REGION Network 26: U201 - ROTAZIONE + CM
   // "U201_OFF1"/"U201_OFF3"
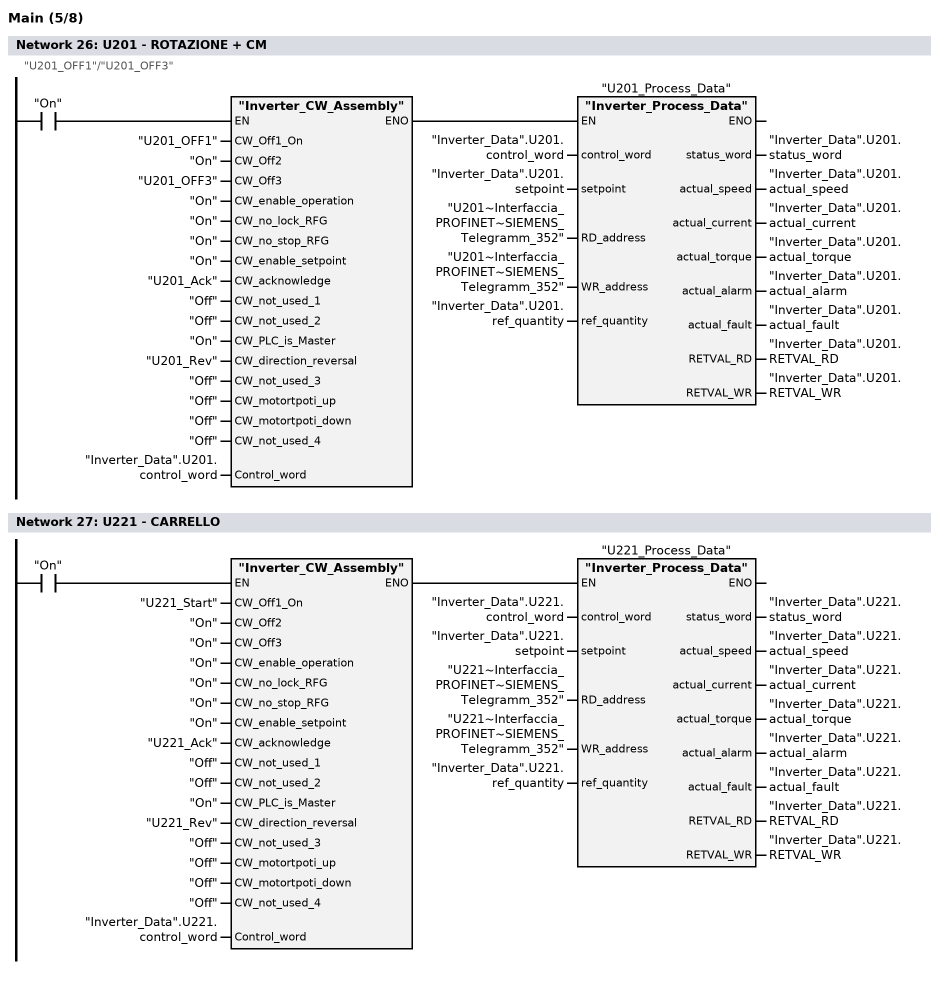
   RUNG wire#powerrail
      Contact( "On" )
      "Inverter_CW_Assembly"(CW_Off1_On := "U201_OFF1", CW_Off2 := "On", CW_Off3 := "U201_OFF3", CW_enable_operation := "On", CW_no_lock_RFG := "On", CW_no_stop_RFG := "On", CW_enable_setpoint := "On", CW_acknowledge := "U201_Ack", CW_not_used_1 := "Off", CW_not_used_2 := "Off", CW_PLC_is_Master := "On", CW_direction_reversal := "U201_Rev", CW_not_used_3 := "Off", CW_motortpoti_up := "Off", CW_motortpoti_down := "Off", CW_not_used_4 := "Off", Control_word := "Inverter_Data".U201.control_word)
      "U201_Process_Data"(control_word := "Inverter_Data".U201.control_word, setpoint := "Inverter_Data".U201.setpoint, RD_address := "U201~Interfaccia_PROFINET~SIEMENS_Telegramm_352", WR_address := "U201~Interfaccia_PROFINET~SIEMENS_Telegramm_352", ref_quantity := "Inverter_Data".U201.ref_quantity, status_word => "Inverter_Data".U201.status_word, actual_speed => "Inverter_Data".U201.actual_speed, actual_current => "Inverter_Data".U201.actual_current, actual_torque => "Inverter_Data".U201.actual_torque, actual_alarm => "Inverter_Data".U201.actual_alarm, actual_fault => "Inverter_Data".U201.actual_fault, RETVAL_RD => "Inverter_Data".U201.RETVAL_RD, RETVAL_WR => "Inverter_Data".U201.RETVAL_WR)
   END_RUNG
   // the same network as SCL:
   "Inverter_CW_Assembly"(EN := "On",
                          CW_Off1_On := "U201_OFF1",
                          CW_Off2 := "On",
                          CW_Off3 := "U201_OFF3",
                          CW_enable_operation := "On",
                          CW_no_lock_RFG := "On",
                          CW_no_stop_RFG := "On",
                          CW_enable_setpoint := "On",
                          CW_acknowledge := "U201_Ack",
                          CW_not_used_1 := "Off",
                          CW_not_used_2 := "Off",
                          CW_PLC_is_Master := "On",
                          CW_direction_reversal := "U201_Rev",
                          CW_not_used_3 := "Off",
                          CW_motortpoti_up := "Off",
                          CW_motortpoti_down := "Off",
                          CW_not_used_4 := "Off",
                          Control_word := "Inverter_Data".U201.control_word,
                          ENO => #_w1);
   IF #_w1 THEN
       "U201_Process_Data"(control_word := "Inverter_Data".U201.control_word,   // "Inverter_Process_Data"
                           setpoint := "Inverter_Data".U201.setpoint,
                           RD_address := "U201~Interfaccia_PROFINET~SIEMENS_Telegramm_352",
                           WR_address := "U201~Interfaccia_PROFINET~SIEMENS_Telegramm_352",
                           ref_quantity := "Inverter_Data".U201.ref_quantity,
                           status_word => "Inverter_Data".U201.status_word,
                           actual_speed => "Inverter_Data".U201.actual_speed,
                           actual_current => "Inverter_Data".U201.actual_current,
                           actual_torque => "Inverter_Data".U201.actual_torque,
                           actual_alarm => "Inverter_Data".U201.actual_alarm,
                           actual_fault => "Inverter_Data".U201.actual_fault,
                           RETVAL_RD => "Inverter_Data".U201.RETVAL_RD,
                           RETVAL_WR => "Inverter_Data".U201.RETVAL_WR);
   END_IF;
END_REGION

REGION Network 27: U221 - CARRELLO
   RUNG wire#powerrail
      Contact( "On" )
      "Inverter_CW_Assembly"(CW_Off1_On := "U221_Start", CW_Off2 := "On", CW_Off3 := "On", CW_enable_operation := "On", CW_no_lock_RFG := "On", CW_no_stop_RFG := "On", CW_enable_setpoint := "On", CW_acknowledge := "U221_Ack", CW_not_used_1 := "Off", CW_not_used_2 := "Off", CW_PLC_is_Master := "On", CW_direction_reversal := "U221_Rev", CW_not_used_3 := "Off", CW_motortpoti_up := "Off", CW_motortpoti_down := "Off", CW_not_used_4 := "Off", Control_word := "Inverter_Data".U221.control_word)
      "U221_Process_Data"(control_word := "Inverter_Data".U221.control_word, setpoint := "Inverter_Data".U221.setpoint, RD_address := "U221~Interfaccia_PROFINET~SIEMENS_Telegramm_352", WR_address := "U221~Interfaccia_PROFINET~SIEMENS_Telegramm_352", ref_quantity := "Inverter_Data".U221.ref_quantity, status_word => "Inverter_Data".U221.status_word, actual_speed => "Inverter_Data".U221.actual_speed, actual_current => "Inverter_Data".U221.actual_current, actual_torque => "Inverter_Data".U221.actual_torque, actual_alarm => "Inverter_Data".U221.actual_alarm, actual_fault => "Inverter_Data".U221.actual_fault, RETVAL_RD => "Inverter_Data".U221.RETVAL_RD, RETVAL_WR => "Inverter_Data".U221.RETVAL_WR)
   END_RUNG
   // the same network as SCL:
   "Inverter_CW_Assembly"(EN := "On",
                          CW_Off1_On := "U221_Start",
                          CW_Off2 := "On",
                          CW_Off3 := "On",
                          CW_enable_operation := "On",
                          CW_no_lock_RFG := "On",
                          CW_no_stop_RFG := "On",
                          CW_enable_setpoint := "On",
                          CW_acknowledge := "U221_Ack",
                          CW_not_used_1 := "Off",
                          CW_not_used_2 := "Off",
                          CW_PLC_is_Master := "On",
                          CW_direction_reversal := "U221_Rev",
                          CW_not_used_3 := "Off",
                          CW_motortpoti_up := "Off",
                          CW_motortpoti_down := "Off",
                          CW_not_used_4 := "Off",
                          Control_word := "Inverter_Data".U221.control_word,
                          ENO => #_w1);
   IF #_w1 THEN
       "U221_Process_Data"(control_word := "Inverter_Data".U221.control_word,   // "Inverter_Process_Data"
                           setpoint := "Inverter_Data".U221.setpoint,
                           RD_address := "U221~Interfaccia_PROFINET~SIEMENS_Telegramm_352",
                           WR_address := "U221~Interfaccia_PROFINET~SIEMENS_Telegramm_352",
                           ref_quantity := "Inverter_Data".U221.ref_quantity,
                           status_word => "Inverter_Data".U221.status_word,
                           actual_speed => "Inverter_Data".U221.actual_speed,
                           actual_current => "Inverter_Data".U221.actual_current,
                           actual_torque => "Inverter_Data".U221.actual_torque,
                           actual_alarm => "Inverter_Data".U221.actual_alarm,
                           actual_fault => "Inverter_Data".U221.actual_fault,
                           RETVAL_RD => "Inverter_Data".U221.RETVAL_RD,
                           RETVAL_WR => "Inverter_Data".U221.RETVAL_WR);
   END_IF;
END_REGION

REGION Network 28: U241 - PRESTIRO (VELOCE)
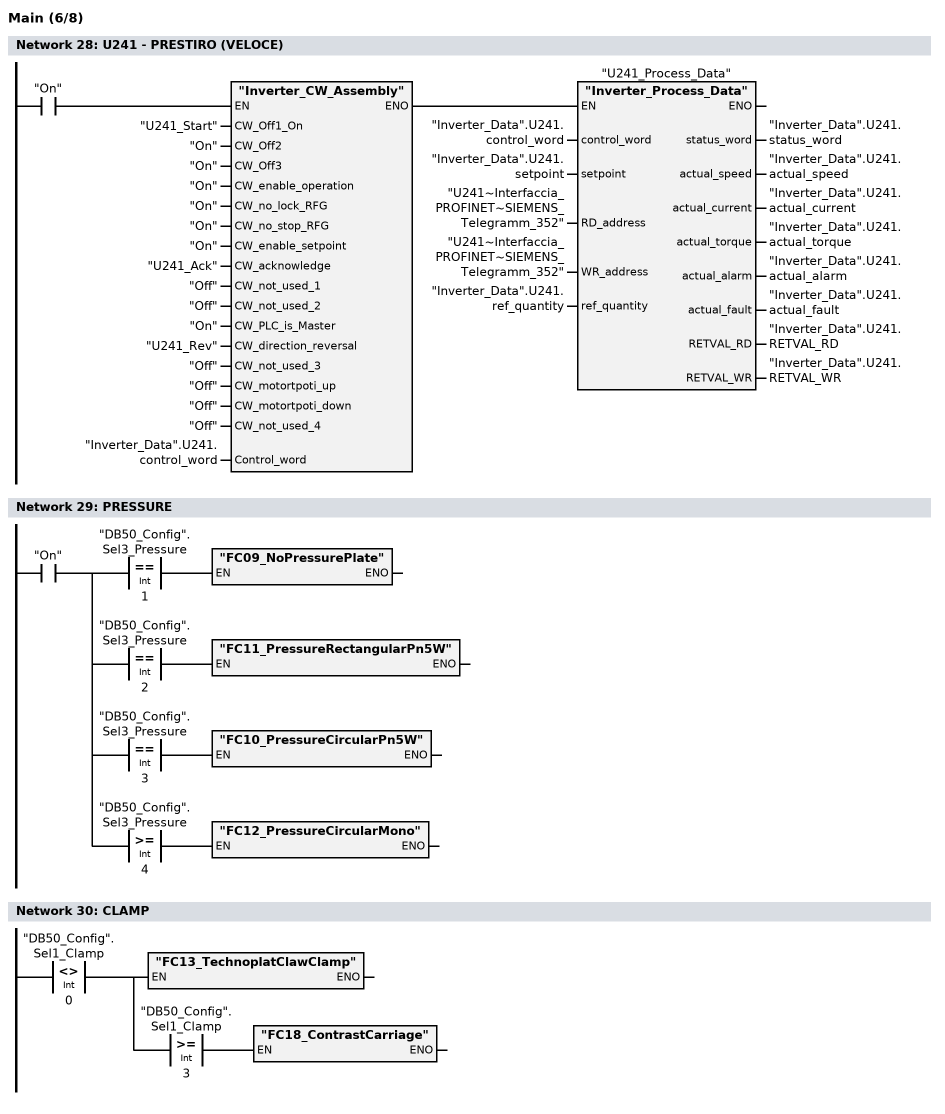
   RUNG wire#powerrail
      Contact( "On" )
      "Inverter_CW_Assembly"(CW_Off1_On := "U241_Start", CW_Off2 := "On", CW_Off3 := "On", CW_enable_operation := "On", CW_no_lock_RFG := "On", CW_no_stop_RFG := "On", CW_enable_setpoint := "On", CW_acknowledge := "U241_Ack", CW_not_used_1 := "Off", CW_not_used_2 := "Off", CW_PLC_is_Master := "On", CW_direction_reversal := "U241_Rev", CW_not_used_3 := "Off", CW_motortpoti_up := "Off", CW_motortpoti_down := "Off", CW_not_used_4 := "Off", Control_word := "Inverter_Data".U241.control_word)
      "U241_Process_Data"(control_word := "Inverter_Data".U241.control_word, setpoint := "Inverter_Data".U241.setpoint, RD_address := "U241~Interfaccia_PROFINET~SIEMENS_Telegramm_352", WR_address := "U241~Interfaccia_PROFINET~SIEMENS_Telegramm_352", ref_quantity := "Inverter_Data".U241.ref_quantity, status_word => "Inverter_Data".U241.status_word, actual_speed => "Inverter_Data".U241.actual_speed, actual_current => "Inverter_Data".U241.actual_current, actual_torque => "Inverter_Data".U241.actual_torque, actual_alarm => "Inverter_Data".U241.actual_alarm, actual_fault => "Inverter_Data".U241.actual_fault, RETVAL_RD => "Inverter_Data".U241.RETVAL_RD, RETVAL_WR => "Inverter_Data".U241.RETVAL_WR)
   END_RUNG
   // the same network as SCL:
   "Inverter_CW_Assembly"(EN := "On",
                          CW_Off1_On := "U241_Start",
                          CW_Off2 := "On",
                          CW_Off3 := "On",
                          CW_enable_operation := "On",
                          CW_no_lock_RFG := "On",
                          CW_no_stop_RFG := "On",
                          CW_enable_setpoint := "On",
                          CW_acknowledge := "U241_Ack",
                          CW_not_used_1 := "Off",
                          CW_not_used_2 := "Off",
                          CW_PLC_is_Master := "On",
                          CW_direction_reversal := "U241_Rev",
                          CW_not_used_3 := "Off",
                          CW_motortpoti_up := "Off",
                          CW_motortpoti_down := "Off",
                          CW_not_used_4 := "Off",
                          Control_word := "Inverter_Data".U241.control_word,
                          ENO => #_w1);
   IF #_w1 THEN
       "U241_Process_Data"(control_word := "Inverter_Data".U241.control_word,   // "Inverter_Process_Data"
                           setpoint := "Inverter_Data".U241.setpoint,
                           RD_address := "U241~Interfaccia_PROFINET~SIEMENS_Telegramm_352",
                           WR_address := "U241~Interfaccia_PROFINET~SIEMENS_Telegramm_352",
                           ref_quantity := "Inverter_Data".U241.ref_quantity,
                           status_word => "Inverter_Data".U241.status_word,
                           actual_speed => "Inverter_Data".U241.actual_speed,
                           actual_current => "Inverter_Data".U241.actual_current,
                           actual_torque => "Inverter_Data".U241.actual_torque,
                           actual_alarm => "Inverter_Data".U241.actual_alarm,
                           actual_fault => "Inverter_Data".U241.actual_fault,
                           RETVAL_RD => "Inverter_Data".U241.RETVAL_RD,
                           RETVAL_WR => "Inverter_Data".U241.RETVAL_WR);
   END_IF;
END_REGION

REGION Network 29: PRESSURE
   RUNG wire#powerrail
      Contact( "On" )
      wire#w1
      { S7_Templates := "SrcType := Int" } EQ_Contact(in1 := "DB50_Config".Sel3_Pressure, in2 := 1)
      "FC09_NoPressurePlate"()
   END_RUNG
   RUNG wire#w1
      { S7_Templates := "SrcType := Int" } EQ_Contact(in1 := "DB50_Config".Sel3_Pressure, in2 := 2)
      "FC11_PressureRectangularPn5W"()
   END_RUNG
   RUNG wire#w1
      { S7_Templates := "SrcType := Int" } EQ_Contact(in1 := "DB50_Config".Sel3_Pressure, in2 := 3)
      "FC10_PressureCircularPn5W"()
   END_RUNG
   RUNG wire#w1
      { S7_Templates := "SrcType := Int" } GE_Contact(in1 := "DB50_Config".Sel3_Pressure, in2 := 4)
      "FC12_PressureCircularMono"()
   END_RUNG
   // the same network as SCL:
   #_w1 := "On";
   IF "On" AND ("DB50_Config".Sel3_Pressure = 1) THEN "FC09_NoPressurePlate"(); END_IF;
   IF #_w1 AND ("DB50_Config".Sel3_Pressure = 2) THEN "FC11_PressureRectangularPn5W"(); END_IF;
   IF #_w1 AND ("DB50_Config".Sel3_Pressure = 3) THEN "FC10_PressureCircularPn5W"(); END_IF;
   IF #_w1 AND ("DB50_Config".Sel3_Pressure >= 4) THEN "FC12_PressureCircularMono"(); END_IF;
END_REGION

REGION Network 30: CLAMP
   RUNG wire#powerrail
      { S7_Templates := "SrcType := Int" } NE_Contact(in1 := "DB50_Config".Sel1_Clamp, in2 := 0)
      wire#w1
      "FC13_TechnoplatClawClamp"()
   END_RUNG
   RUNG wire#w1
      { S7_Templates := "SrcType := Int" } GE_Contact(in1 := "DB50_Config".Sel1_Clamp, in2 := 3)
      "FC18_ContrastCarriage"()
   END_RUNG
   // the same network as SCL:
   #_w1 := "DB50_Config".Sel1_Clamp <> 0;
   IF #_w1 THEN "FC13_TechnoplatClawClamp"(); END_IF;
   IF #_w1 AND ("DB50_Config".Sel1_Clamp >= 3) THEN "FC18_ContrastCarriage"(); END_IF;
END_REGION

REGION Network 31: Lifter selection
END_REGION

REGION Network 32: TOP
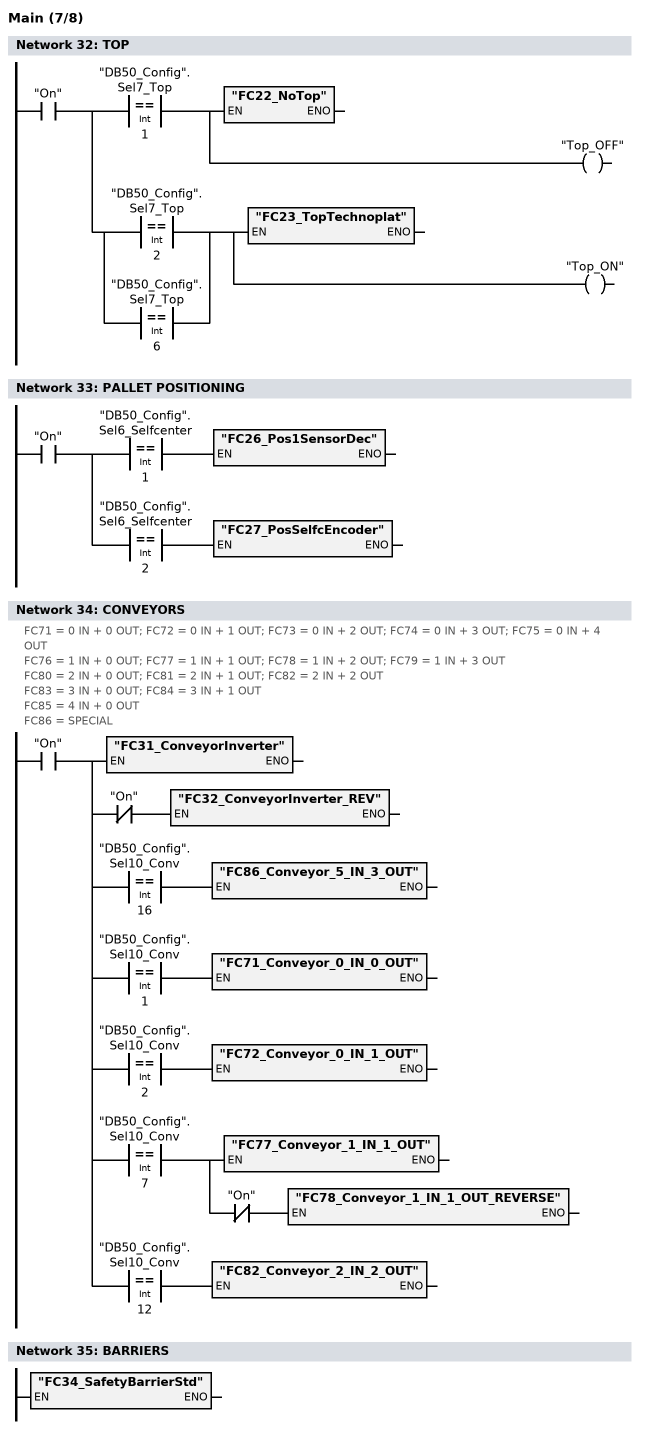
   RUNG wire#powerrail
      Contact( "On" )
      wire#w1
      { S7_Templates := "SrcType := Int" } EQ_Contact(in1 := "DB50_Config".Sel7_Top, in2 := 1)
      wire#w2
      "FC22_NoTop"()
   END_RUNG
   RUNG wire#w2
      Coil( "Top_OFF" )
   END_RUNG
   RUNG wire#w1
      { S7_Templates := "SrcType := Int" } EQ_Contact(in1 := "DB50_Config".Sel7_Top, in2 := 2)
      wire#w3
      "FC23_TopTechnoplat"()
   END_RUNG
   RUNG wire#w1
      { S7_Templates := "SrcType := Int" } EQ_Contact(in1 := "DB50_Config".Sel7_Top, in2 := 6)
   END_RUNG wire#w3
   RUNG wire#w3
      Coil( "Top_ON" )
   END_RUNG
   // the same network as SCL:
   #_w1 := "On" AND ("DB50_Config".Sel7_Top = 1);
   #_w2 := "On";
   IF #_w1 THEN "FC22_NoTop"(); END_IF;
   "Top_OFF" := #_w1;
   #_w3 := #_w2 AND (("DB50_Config".Sel7_Top = 2) OR ("DB50_Config".Sel7_Top = 6));
   IF #_w3 THEN "FC23_TopTechnoplat"(); END_IF;
   "Top_ON" := #_w3;
END_REGION

REGION Network 33: PALLET POSITIONING
   RUNG wire#powerrail
      Contact( "On" )
      wire#w1
      { S7_Templates := "SrcType := Int" } EQ_Contact(in1 := "DB50_Config".Sel6_Selfcenter, in2 := 1)
      "FC26_Pos1SensorDec"()
   END_RUNG
   RUNG wire#w1
      { S7_Templates := "SrcType := Int" } EQ_Contact(in1 := "DB50_Config".Sel6_Selfcenter, in2 := 2)
      "FC27_PosSelfcEncoder"()
   END_RUNG
   // the same network as SCL:
   #_w1 := "On";
   IF "On" AND ("DB50_Config".Sel6_Selfcenter = 1) THEN "FC26_Pos1SensorDec"(); END_IF;
   IF #_w1 AND ("DB50_Config".Sel6_Selfcenter = 2) THEN "FC27_PosSelfcEncoder"(); END_IF;
END_REGION

REGION Network 34: CONVEYORS
   // FC71 = 0 IN + 0 OUT; FC72 = 0 IN + 1 OUT; FC73 = 0 IN + 2 OUT; FC74 = 0 IN + 3 OUT; FC75 = 0 IN + 4 OUT
   // FC76 = 1 IN + 0 OUT; FC77 = 1 IN + 1 OUT; FC78 = 1 IN + 2 OUT; FC79 = 1 IN + 3 OUT
   // FC80 = 2 IN + 0 OUT; FC81 = 2 IN + 1 OUT; FC82 = 2 IN + 2 OUT
   // FC83 = 3 IN + 0 OUT; FC84 = 3 IN + 1 OUT
   // FC85 = 4 IN + 0 OUT
   // FC86 = SPECIAL
   RUNG wire#powerrail
      Contact( "On" )
      wire#w1
      "FC31_ConveyorInverter"()
   END_RUNG
   RUNG wire#w1
      I_Contact( "On" )
      "FC32_ConveyorInverter_REV"()
   END_RUNG
   RUNG wire#w1
      { S7_Templates := "SrcType := Int" } EQ_Contact(in1 := "DB50_Config".Sel10_Conv, in2 := 16)
      "FC86_Conveyor_5_IN_3_OUT"()
   END_RUNG
   RUNG wire#w1
      { S7_Templates := "SrcType := Int" } EQ_Contact(in1 := "DB50_Config".Sel10_Conv, in2 := 1)
      "FC71_Conveyor_0_IN_0_OUT"()
   END_RUNG
   RUNG wire#w1
      { S7_Templates := "SrcType := Int" } EQ_Contact(in1 := "DB50_Config".Sel10_Conv, in2 := 2)
      "FC72_Conveyor_0_IN_1_OUT"()
   END_RUNG
   RUNG wire#w1
      { S7_Templates := "SrcType := Int" } EQ_Contact(in1 := "DB50_Config".Sel10_Conv, in2 := 7)
      wire#w2
      "FC77_Conveyor_1_IN_1_OUT"()
   END_RUNG
   RUNG wire#w2
      I_Contact( "On" )
      "FC78_Conveyor_1_IN_1_OUT_REVERSE"()
   END_RUNG
   RUNG wire#w1
      { S7_Templates := "SrcType := Int" } EQ_Contact(in1 := "DB50_Config".Sel10_Conv, in2 := 12)
      "FC82_Conveyor_2_IN_2_OUT"()
   END_RUNG
   // the same network as SCL:
   #_w1 := "On";
   IF #_w1 THEN "FC31_ConveyorInverter"(); END_IF;
   IF #_w1 AND NOT "On" THEN "FC32_ConveyorInverter_REV"(); END_IF;
   IF #_w1 AND ("DB50_Config".Sel10_Conv = 16) THEN "FC86_Conveyor_5_IN_3_OUT"(); END_IF;
   IF #_w1 AND ("DB50_Config".Sel10_Conv = 1) THEN "FC71_Conveyor_0_IN_0_OUT"(); END_IF;
   IF #_w1 AND ("DB50_Config".Sel10_Conv = 2) THEN "FC72_Conveyor_0_IN_1_OUT"(); END_IF;
   #_w2 := #_w1 AND ("DB50_Config".Sel10_Conv = 7);
   IF #_w2 THEN "FC77_Conveyor_1_IN_1_OUT"(); END_IF;
   IF #_w2 AND NOT "On" THEN "FC78_Conveyor_1_IN_1_OUT_REVERSE"(); END_IF;
   IF #_w1 AND ("DB50_Config".Sel10_Conv = 12) THEN "FC82_Conveyor_2_IN_2_OUT"(); END_IF;
END_REGION

REGION Network 35: BARRIERS
   RUNG wire#powerrail
      "FC34_SafetyBarrierStd"()
   END_RUNG
   // the same network as SCL:
   "FC34_SafetyBarrierStd"();
END_REGION

REGION Network 36: MULTIPROGRAM
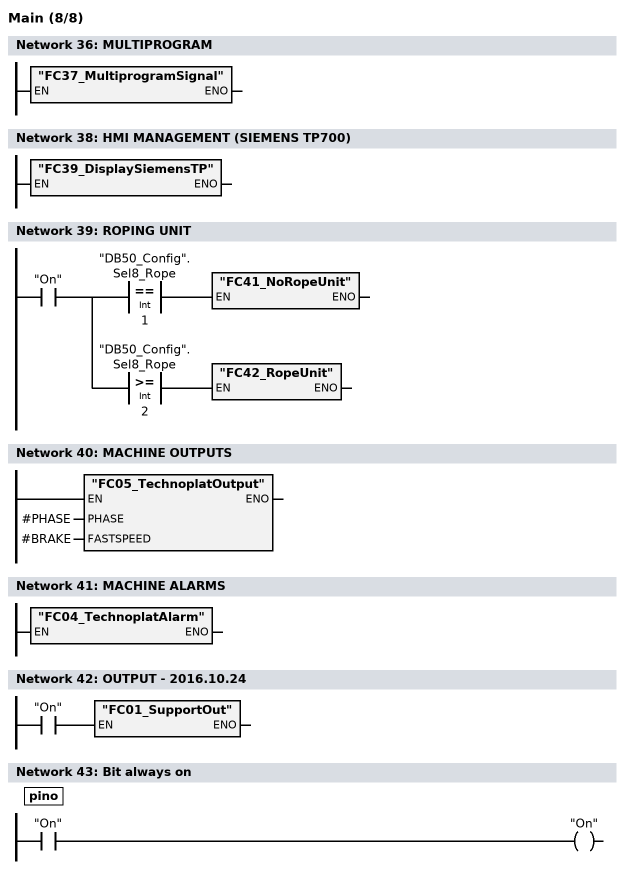
   RUNG wire#powerrail
      "FC37_MultiprogramSignal"()
   END_RUNG
   // the same network as SCL:
   "FC37_MultiprogramSignal"();
END_REGION

REGION Network 37: Incomplete pallet
END_REGION

REGION Network 38: HMI MANAGEMENT (SIEMENS TP700)
   RUNG wire#powerrail
      "FC39_DisplaySiemensTP"()
   END_RUNG
   // the same network as SCL:
   "FC39_DisplaySiemensTP"();
END_REGION

REGION Network 39: ROPING UNIT
   RUNG wire#powerrail
      Contact( "On" )
      wire#w1
      { S7_Templates := "SrcType := Int" } EQ_Contact(in1 := "DB50_Config".Sel8_Rope, in2 := 1)
      "FC41_NoRopeUnit"()
   END_RUNG
   RUNG wire#w1
      { S7_Templates := "SrcType := Int" } GE_Contact(in1 := "DB50_Config".Sel8_Rope, in2 := 2)
      "FC42_RopeUnit"()
   END_RUNG
   // the same network as SCL:
   #_w1 := "On";
   IF "On" AND ("DB50_Config".Sel8_Rope = 1) THEN "FC41_NoRopeUnit"(); END_IF;
   IF #_w1 AND ("DB50_Config".Sel8_Rope >= 2) THEN "FC42_RopeUnit"(); END_IF;
END_REGION

REGION Network 40: MACHINE OUTPUTS
   RUNG wire#powerrail
      "FC05_TechnoplatOutput"(PHASE := #PHASE, FASTSPEED := #BRAKE)
   END_RUNG
   // the same network as SCL:
   "FC05_TechnoplatOutput"(PHASE := #PHASE, FASTSPEED := #BRAKE);
END_REGION

REGION Network 41: MACHINE ALARMS
   RUNG wire#powerrail
      "FC04_TechnoplatAlarm"()
   END_RUNG
   // the same network as SCL:
   "FC04_TechnoplatAlarm"();
END_REGION

REGION Network 42: OUTPUT - 2016.10.24
   RUNG wire#powerrail
      Contact( "On" )
      "FC01_SupportOut"()
   END_RUNG
   // the same network as SCL:
   IF "On" THEN "FC01_SupportOut"(); END_IF;
END_REGION

REGION Network 43: Bit always on
   Label( pino )
   RUNG wire#powerrail
      Contact( "On" )
      Coil( "On" )
   END_RUNG
   // the same network as SCL:
   pino:
   "On" := "On";
END_REGION
END_ORGANIZATION_BLOCK

FUNCTION_BLOCK "Modbus"   // FB20, FBD
{ S7_Optimized_Access := 'FALSE' }
VERSION : 0.1
// stored: AutoNumber false, IsIECCheckEnabled false, SetENOAutomatically false, UDAEnableTagReadback false
   VAR_INPUT
      BAUDRATE : UDInt := 115200;
      HW_ID : PORT := 272;
      RESP_TO : UInt := 1000;
      CYCLIC_PROCESSING : Bool := true;
      MB_ADDR : UInt := 8;
      DATA_AD_R : UDInt := 40001;
      DATA_AD_W : UDInt := 40006;
      DATA_LEN_R : UInt := 5;
      DATA_LEN_W : UInt := 5;
      ReadOnly : Bool := 1;   // Read only (1)
   END_VAR
   VAR_OUTPUT
      ERROR : Bool;
      ERROR_INFO : Struct
         drive_number : USInt;
         "step" : USInt;
         STATUS : Word;
      END_STRUCT;
   END_VAR
   VAR_IN_OUT
      ReadDone_0 : Bool;   // Read done for prestretch board (1)
      DT_PTR_IN : Variant;
      DT_PTR_OUT : Variant;
   END_VAR
   VAR DB_SPECIFIC
      drive_index : USInt := 1;
      "step" : USInt := 0;
      REQ : Bool;
      extended_restart : Bool;
      start_internal : Bool;
   END_VAR
   VAR
      MB_COMM_LOAD_Instance { S7_SetPoint := 'True'} : MB_COMM_LOAD;
      MB_MASTER_Instance { S7_SetPoint := 'True'} : MB_MASTER;
   END_VAR
   VAR_TEMP
      _DONE : Bool;
      _ERROR : Bool;
      _STATUS : Word;
      _cyclic_processing : Bool;
   END_VAR
   VAR_TEMP   // added for the SCL form of the ladder/FBD networks
      _w1 : Bool;
      _w2 : Bool;
      _w3 : Bool;
   END_VAR
BEGIN

REGION Network 1: First cycle
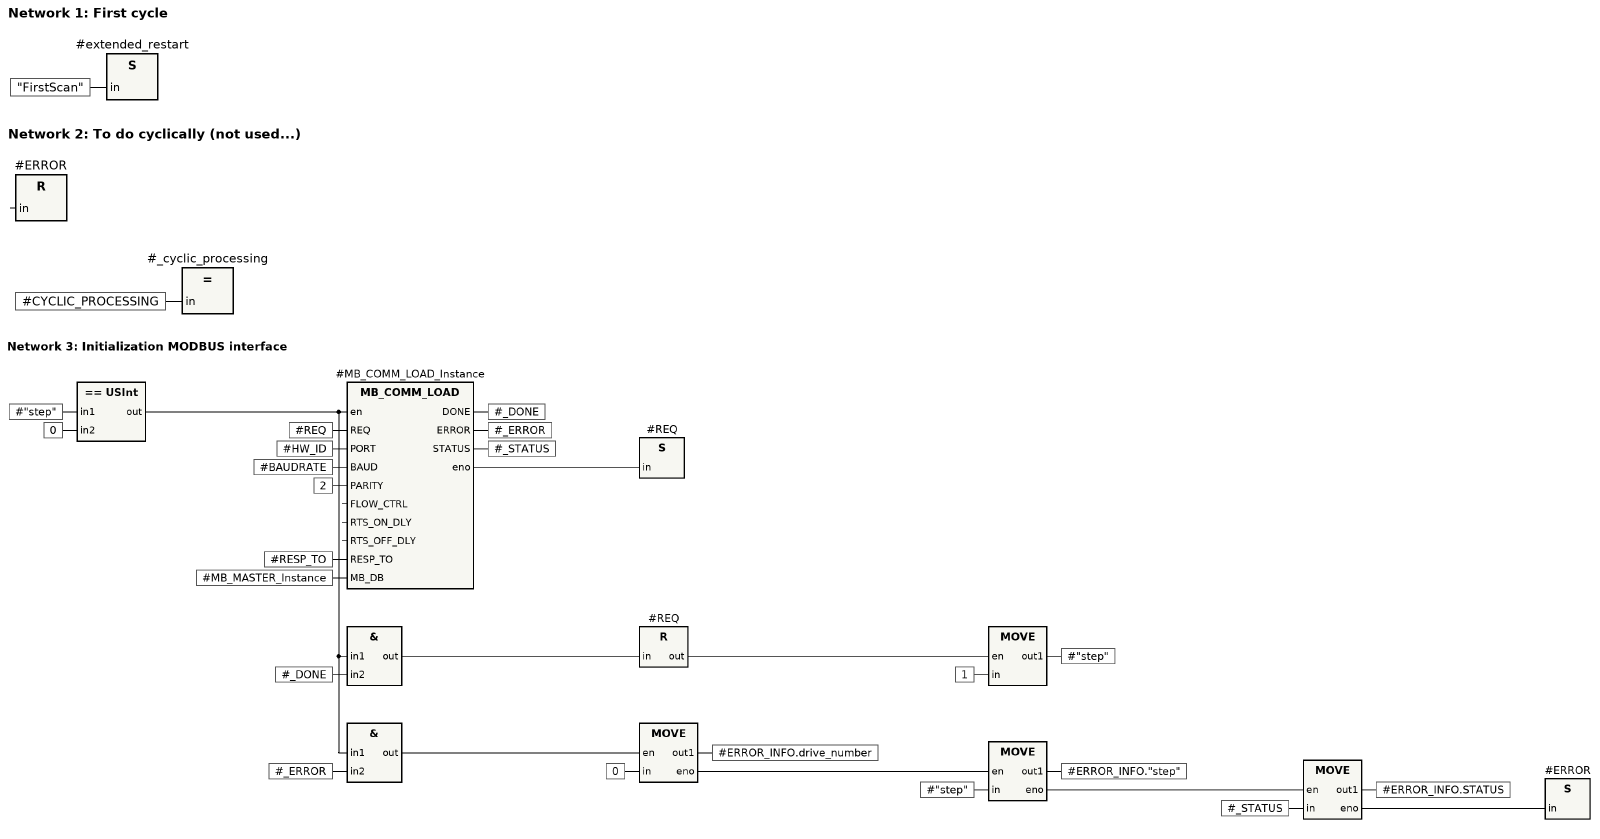
   IF "FirstScan" THEN #extended_restart := TRUE; END_IF;
END_REGION

REGION Network 2: To do cyclically (not used...)
   #ERROR := FALSE;
   #_cyclic_processing := #CYCLIC_PROCESSING;
END_REGION

REGION Network 3: Initialization MODBUS interface
   // ENO of a box is taken as its EN; it also drops when the box reports an error
   #_w1 := #"step" = 0;
   #MB_COMM_LOAD_Instance(EN := #_w1,   // MB_COMM_LOAD
                          REQ := #REQ,
                          PORT := #HW_ID,
                          BAUD := #BAUDRATE,
                          PARITY := 2,
                          RESP_TO := #RESP_TO,
                          MB_DB := #MB_MASTER_Instance,
                          DONE => #_DONE,
                          ERROR => #_ERROR,
                          STATUS => #_STATUS,
                          ENO => #_w2);
   IF #_w2 THEN #REQ := TRUE; END_IF;
   IF #_w1 AND #_DONE THEN
       #REQ := FALSE;
       #"step" := 1;
   END_IF;
   IF #_w1 AND #_ERROR THEN
       #ERROR_INFO.drive_number := 0;
       #ERROR_INFO."step" := #"step";
       #ERROR_INFO.STATUS := #_STATUS;
       #ERROR := TRUE;
   END_IF;
END_REGION

REGION Network 4: READ
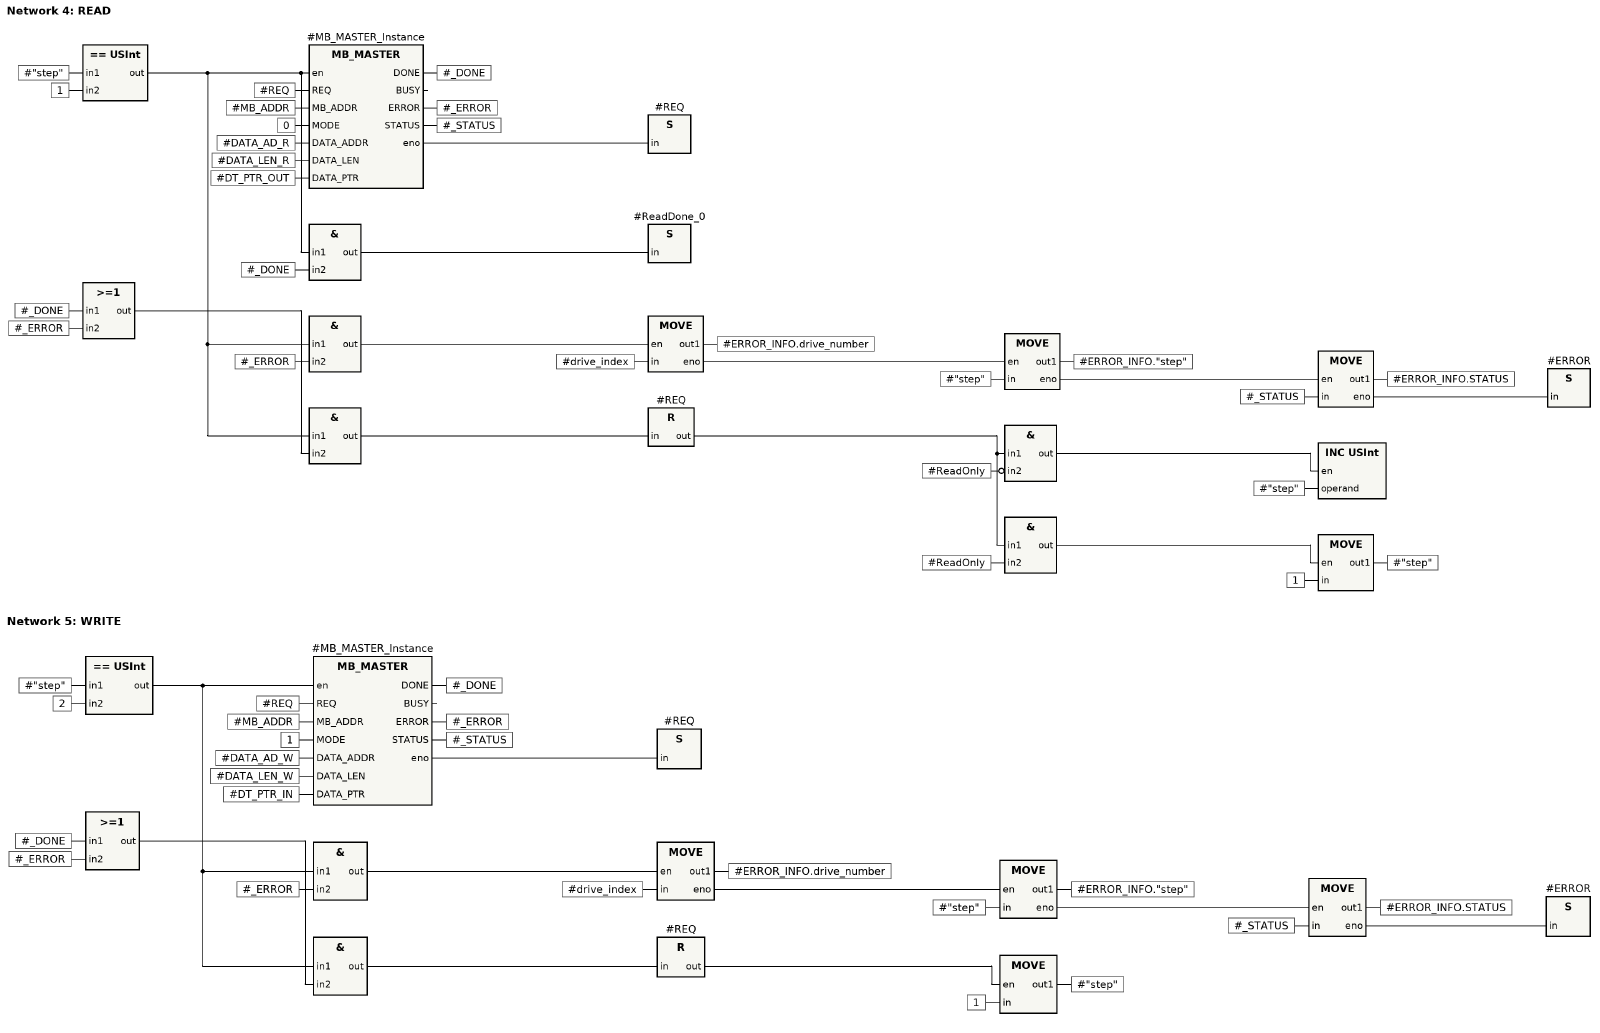
   // ENO of a box is taken as its EN; it also drops when the box reports an error
   #_w1 := #"step" = 1;
   #MB_MASTER_Instance(EN := #_w1,   // MB_MASTER
                       REQ := #REQ,
                       MB_ADDR := #MB_ADDR,
                       MODE := 0,
                       DATA_ADDR := #DATA_AD_R,
                       DATA_LEN := #DATA_LEN_R,
                       DATA_PTR := #DT_PTR_OUT,
                       DONE => #_DONE,
                       ERROR => #_ERROR,
                       STATUS => #_STATUS,
                       ENO => #_w2);
   IF #_w2 THEN #REQ := TRUE; END_IF;
   IF #_w1 AND #_DONE THEN #ReadDone_0 := TRUE; END_IF;
   IF #_w1 AND #_ERROR THEN
       #ERROR_INFO.drive_number := #drive_index;
       #ERROR_INFO."step" := #"step";
       #ERROR_INFO.STATUS := #_STATUS;
       #ERROR := TRUE;
   END_IF;
   #_w3 := #_w1 AND (#_DONE OR #_ERROR);
   IF #_w3 THEN #REQ := FALSE; END_IF;
   IF #_w3 AND NOT #ReadOnly THEN #"step" := #"step" + 1; END_IF;
   IF #_w3 AND #ReadOnly THEN #"step" := 1; END_IF;
END_REGION

REGION Network 5: WRITE
   // ENO of a box is taken as its EN; it also drops when the box reports an error
   #_w1 := #"step" = 2;
   #MB_MASTER_Instance(EN := #_w1,   // MB_MASTER
                       REQ := #REQ,
                       MB_ADDR := #MB_ADDR,
                       MODE := 1,
                       DATA_ADDR := #DATA_AD_W,
                       DATA_LEN := #DATA_LEN_W,
                       DATA_PTR := #DT_PTR_IN,
                       DONE => #_DONE,
                       ERROR => #_ERROR,
                       STATUS => #_STATUS,
                       ENO => #_w2);
   IF #_w2 THEN #REQ := TRUE; END_IF;
   IF #_w1 AND #_ERROR THEN
       #ERROR_INFO.drive_number := #drive_index;
       #ERROR_INFO."step" := #"step";
       #ERROR_INFO.STATUS := #_STATUS;
       #ERROR := TRUE;
   END_IF;
   IF #_w1 AND (#_DONE OR #_ERROR) THEN
       #REQ := FALSE;
       #"step" := 1;
   END_IF;
END_REGION
END_FUNCTION_BLOCK

FUNCTION "FC00_SupportIn" : Void   // FC0, LAD
TITLE = Input support memory
{ S7_Optimized_Access := 'FALSE' }
AUTHOR : Robopac
VERSION : 0.0
// stored: AutoNumber false, IsIECCheckEnabled false, SetENOAutomatically false, UDAEnableTagReadback false
   VAR_TEMP
      AC1 : Int;
      AC2 : Int;
   END_VAR
BEGIN

REGION Network 1: STANDARD
END_REGION

REGION Network 2: Pressure switch (Technoplat)
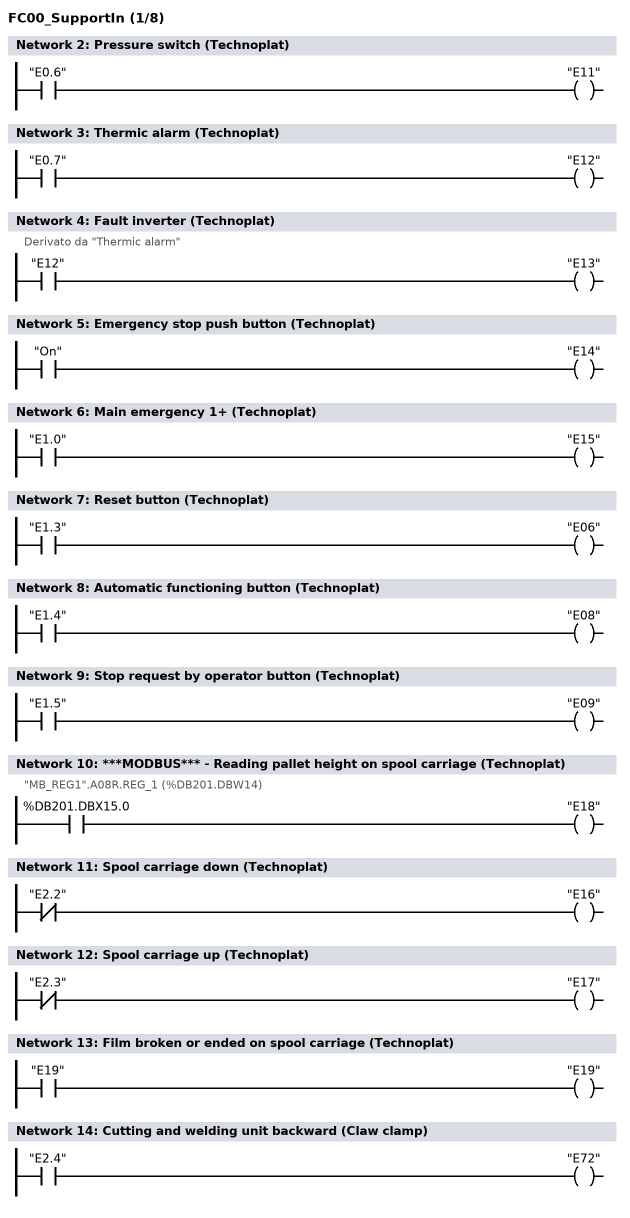
   RUNG wire#powerrail
      Contact( "E0.6" )
      Coil( "E11" )
   END_RUNG
   // the same network as SCL:
   "E11" := "E0.6";
END_REGION

REGION Network 3: Thermic alarm (Technoplat)
   RUNG wire#powerrail
      Contact( "E0.7" )
      Coil( "E12" )
   END_RUNG
   // the same network as SCL:
   "E12" := "E0.7";
END_REGION

REGION Network 4: Fault inverter (Technoplat)
   // Derivato da "Thermic alarm"
   RUNG wire#powerrail
      Contact( "E12" )
      Coil( "E13" )
   END_RUNG
   // the same network as SCL:
   "E13" := "E12";
END_REGION

REGION Network 5: Emergency stop push button (Technoplat)
   RUNG wire#powerrail
      Contact( "On" )
      Coil( "E14" )
   END_RUNG
   // the same network as SCL:
   "E14" := "On";
END_REGION

REGION Network 6: Main emergency 1+ (Technoplat)
   RUNG wire#powerrail
      Contact( "E1.0" )
      Coil( "E15" )
   END_RUNG
   // the same network as SCL:
   "E15" := "E1.0";
END_REGION

REGION Network 7: Reset button (Technoplat)
   RUNG wire#powerrail
      Contact( "E1.3" )
      Coil( "E06" )
   END_RUNG
   // the same network as SCL:
   "E06" := "E1.3";
END_REGION

REGION Network 8: Automatic functioning button (Technoplat)
   RUNG wire#powerrail
      Contact( "E1.4" )
      Coil( "E08" )
   END_RUNG
   // the same network as SCL:
   "E08" := "E1.4";
END_REGION

REGION Network 9: Stop request by operator button (Technoplat)
   RUNG wire#powerrail
      Contact( "E1.5" )
      Coil( "E09" )
   END_RUNG
   // the same network as SCL:
   "E09" := "E1.5";
END_REGION

REGION Network 10: ***MODBUS*** - Reading pallet height on spool carriage (Technoplat)
   // "MB_REG1".A08R.REG_1 (%DB201.DBW14)
   RUNG wire#powerrail
      Contact( %DB201.DBX15.0 )
      Coil( "E18" )
   END_RUNG
   // the same network as SCL:
   "E18" := %DB201.DBX15.0;
END_REGION

REGION Network 11: Spool carriage down (Technoplat)
   RUNG wire#powerrail
      I_Contact( "E2.2" )
      Coil( "E16" )
   END_RUNG
   // the same network as SCL:
   "E16" := NOT "E2.2";
END_REGION

REGION Network 12: Spool carriage up (Technoplat)
   RUNG wire#powerrail
      I_Contact( "E2.3" )
      Coil( "E17" )
   END_RUNG
   // the same network as SCL:
   "E17" := NOT "E2.3";
END_REGION

REGION Network 13: Film broken or ended on spool carriage (Technoplat)
   RUNG wire#powerrail
      Contact( "E19" )
      Coil( "E19" )
   END_RUNG
   // the same network as SCL:
   "E19" := "E19";
END_REGION

REGION Network 14: Cutting and welding unit backward (Claw clamp)
   RUNG wire#powerrail
      Contact( "E2.4" )
      Coil( "E72" )
   END_RUNG
   // the same network as SCL:
   "E72" := "E2.4";
END_REGION

REGION Network 15: Cutting and welding unit forward (Claw clamp)
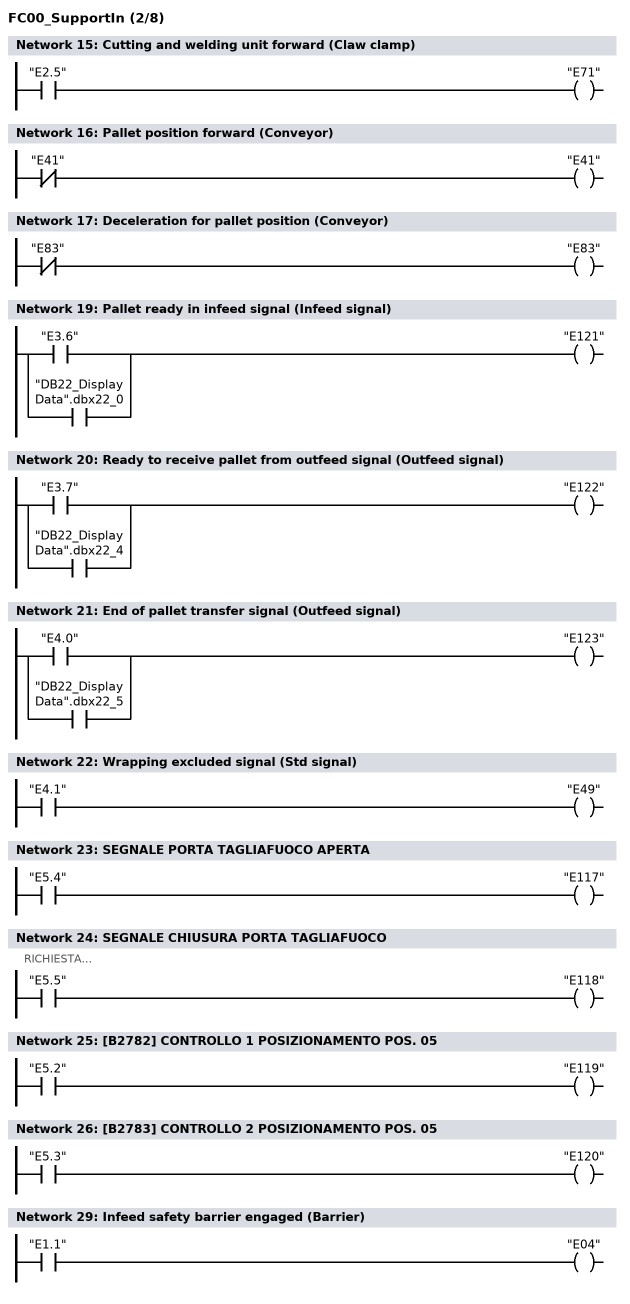
   RUNG wire#powerrail
      Contact( "E2.5" )
      Coil( "E71" )
   END_RUNG
   // the same network as SCL:
   "E71" := "E2.5";
END_REGION

REGION Network 16: Pallet position forward (Conveyor)
   RUNG wire#powerrail
      I_Contact( "E41" )
      Coil( "E41" )
   END_RUNG
   // the same network as SCL:
   "E41" := NOT "E41";
END_REGION

REGION Network 17: Deceleration for pallet position (Conveyor)
   RUNG wire#powerrail
      I_Contact( "E83" )
      Coil( "E83" )
   END_RUNG
   // the same network as SCL:
   "E83" := NOT "E83";
END_REGION

REGION Network 18: EXCHANGE SIGNALS
END_REGION

REGION Network 19: Pallet ready in infeed signal (Infeed signal)
   RUNG wire#powerrail
      Contact( "E3.6" )
      wire#w1
      Coil( "E121" )
   END_RUNG
   RUNG wire#powerrail
      Contact( "DB22_DisplayData".dbx22_0 )
   END_RUNG wire#w1
   // the same network as SCL:
   "E121" := "E3.6" OR "DB22_DisplayData".dbx22_0;
END_REGION

REGION Network 20: Ready to receive pallet from outfeed signal (Outfeed signal)
   RUNG wire#powerrail
      Contact( "E3.7" )
      wire#w1
      Coil( "E122" )
   END_RUNG
   RUNG wire#powerrail
      Contact( "DB22_DisplayData".dbx22_4 )
   END_RUNG wire#w1
   // the same network as SCL:
   "E122" := "E3.7" OR "DB22_DisplayData".dbx22_4;
END_REGION

REGION Network 21: End of pallet transfer signal (Outfeed signal)
   RUNG wire#powerrail
      Contact( "E4.0" )
      wire#w1
      Coil( "E123" )
   END_RUNG
   RUNG wire#powerrail
      Contact( "DB22_DisplayData".dbx22_5 )
   END_RUNG wire#w1
   // the same network as SCL:
   "E123" := "E4.0" OR "DB22_DisplayData".dbx22_5;
END_REGION

REGION Network 22: Wrapping excluded signal (Std signal)
   RUNG wire#powerrail
      Contact( "E4.1" )
      Coil( "E49" )
   END_RUNG
   // the same network as SCL:
   "E49" := "E4.1";
END_REGION

REGION Network 23: SEGNALE PORTA TAGLIAFUOCO APERTA
   RUNG wire#powerrail
      Contact( "E5.4" )
      Coil( "E117" )
   END_RUNG
   // the same network as SCL:
   "E117" := "E5.4";
END_REGION

REGION Network 24: SEGNALE CHIUSURA PORTA TAGLIAFUOCO
   // RICHIESTA...
   RUNG wire#powerrail
      Contact( "E5.5" )
      Coil( "E118" )
   END_RUNG
   // the same network as SCL:
   "E118" := "E5.5";
END_REGION

REGION Network 25: [B2782] CONTROLLO 1 POSIZIONAMENTO POS. 05
   RUNG wire#powerrail
      Contact( "E5.2" )
      Coil( "E119" )
   END_RUNG
   // the same network as SCL:
   "E119" := "E5.2";
END_REGION

REGION Network 26: [B2783] CONTROLLO 2 POSIZIONAMENTO POS. 05
   RUNG wire#powerrail
      Contact( "E5.3" )
      Coil( "E120" )
   END_RUNG
   // the same network as SCL:
   "E120" := "E5.3";
END_REGION

REGION Network 27: ACCESSORIES
END_REGION

REGION Network 28: ***BARRIERS***
END_REGION

REGION Network 29: Infeed safety barrier engaged (Barrier)
   RUNG wire#powerrail
      Contact( "E1.1" )
      Coil( "E04" )
   END_RUNG
   // the same network as SCL:
   "E04" := "E1.1";
END_REGION

REGION Network 30: Outfeed safety barrier engaged (Barrier)
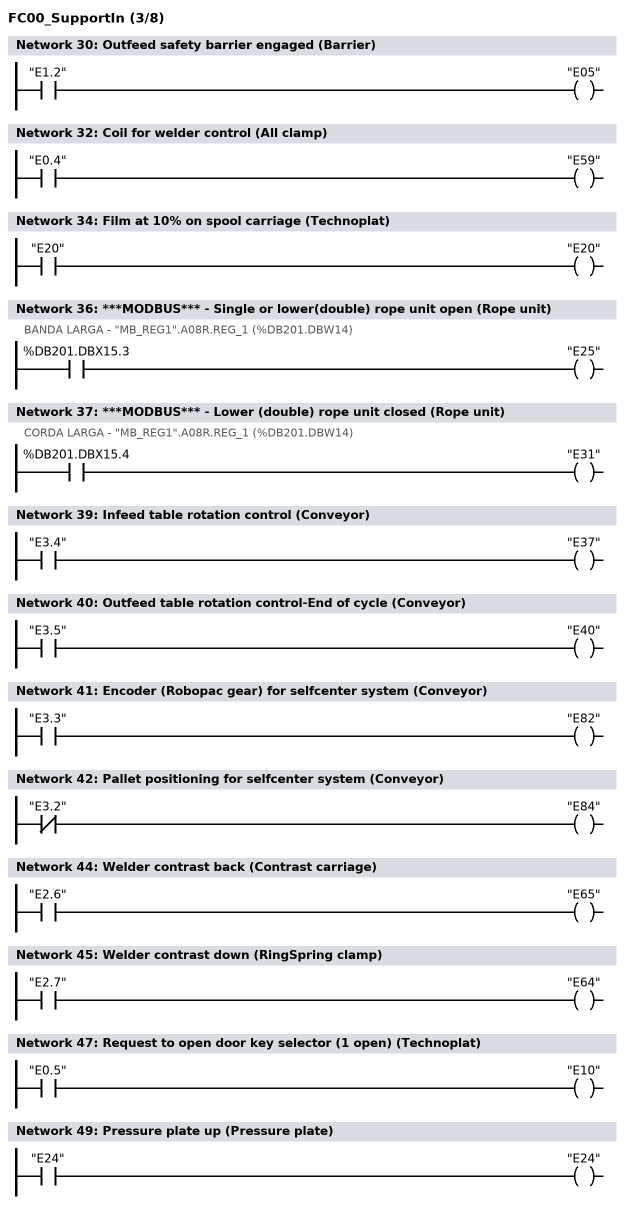
   RUNG wire#powerrail
      Contact( "E1.2" )
      Coil( "E05" )
   END_RUNG
   // the same network as SCL:
   "E05" := "E1.2";
END_REGION

REGION Network 31: ***WELDER***
END_REGION

REGION Network 32: Coil for welder control (All clamp)
   RUNG wire#powerrail
      Contact( "E0.4" )
      Coil( "E59" )
   END_RUNG
   // the same network as SCL:
   "E59" := "E0.4";
END_REGION

REGION Network 33: ***ES_FILM***
END_REGION

REGION Network 34: Film at 10% on spool carriage (Technoplat)
   RUNG wire#powerrail
      Contact( "E20" )
      Coil( "E20" )
   END_RUNG
   // the same network as SCL:
   "E20" := "E20";
END_REGION

REGION Network 35: ***BAND/ROPE***
END_REGION

REGION Network 36: ***MODBUS*** - Single or lower(double) rope unit open (Rope unit)
   // BANDA LARGA - "MB_REG1".A08R.REG_1 (%DB201.DBW14)
   RUNG wire#powerrail
      Contact( %DB201.DBX15.3 )
      Coil( "E25" )
   END_RUNG
   // the same network as SCL:
   "E25" := %DB201.DBX15.3;
END_REGION

REGION Network 37: ***MODBUS*** - Lower (double) rope unit closed (Rope unit)
   // CORDA LARGA - "MB_REG1".A08R.REG_1 (%DB201.DBW14)
   RUNG wire#powerrail
      Contact( %DB201.DBX15.4 )
      Coil( "E31" )
   END_RUNG
   // the same network as SCL:
   "E31" := %DB201.DBX15.4;
END_REGION

REGION Network 38: ***SELF-CENTER***
END_REGION

REGION Network 39: Infeed table rotation control (Conveyor)
   RUNG wire#powerrail
      Contact( "E3.4" )
      Coil( "E37" )
   END_RUNG
   // the same network as SCL:
   "E37" := "E3.4";
END_REGION

REGION Network 40: Outfeed table rotation control-End of cycle (Conveyor)
   RUNG wire#powerrail
      Contact( "E3.5" )
      Coil( "E40" )
   END_RUNG
   // the same network as SCL:
   "E40" := "E3.5";
END_REGION

REGION Network 41: Encoder (Robopac gear) for selfcenter system (Conveyor)
   RUNG wire#powerrail
      Contact( "E3.3" )
      Coil( "E82" )
   END_RUNG
   // the same network as SCL:
   "E82" := "E3.3";
END_REGION

REGION Network 42: Pallet positioning for selfcenter system (Conveyor)
   RUNG wire#powerrail
      I_Contact( "E3.2" )
      Coil( "E84" )
   END_RUNG
   // the same network as SCL:
   "E84" := NOT "E3.2";
END_REGION

REGION Network 43: ***CONTRAST***
END_REGION

REGION Network 44: Welder contrast back (Contrast carriage)
   RUNG wire#powerrail
      Contact( "E2.6" )
      Coil( "E65" )
   END_RUNG
   // the same network as SCL:
   "E65" := "E2.6";
END_REGION

REGION Network 45: Welder contrast down (RingSpring clamp)
   RUNG wire#powerrail
      Contact( "E2.7" )
      Coil( "E64" )
   END_RUNG
   // the same network as SCL:
   "E64" := "E2.7";
END_REGION

REGION Network 46: ***DOOR***
END_REGION

REGION Network 47: Request to open door key selector (1 open) (Technoplat)
   RUNG wire#powerrail
      Contact( "E0.5" )
      Coil( "E10" )
   END_RUNG
   // the same network as SCL:
   "E10" := "E0.5";
END_REGION

REGION Network 48: ***PRESSURE***
END_REGION

REGION Network 49: Pressure plate up (Pressure plate)
   RUNG wire#powerrail
      Contact( "E24" )
      Coil( "E24" )
   END_RUNG
   // the same network as SCL:
   "E24" := "E24";
END_REGION

REGION Network 50: Pressure plate positioning
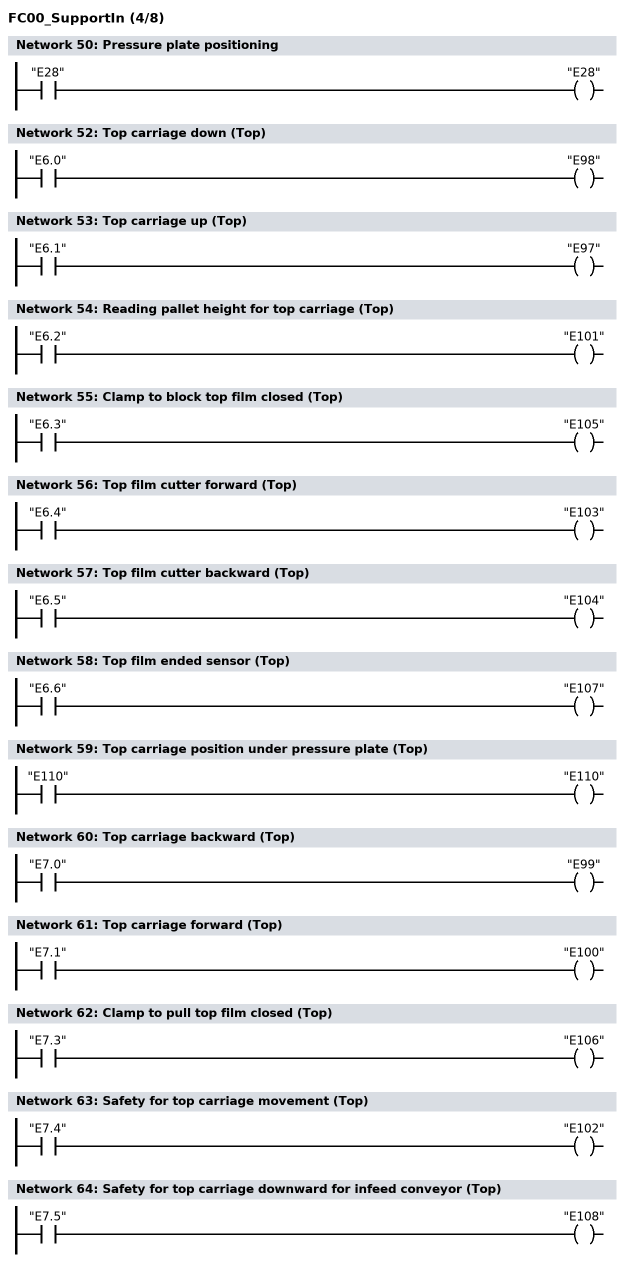
   RUNG wire#powerrail
      Contact( "E28" )
      Coil( "E28" )
   END_RUNG
   // the same network as SCL:
   "E28" := "E28";
END_REGION

REGION Network 51: ***TOP***
END_REGION

REGION Network 52: Top carriage down (Top)
   RUNG wire#powerrail
      Contact( "E6.0" )
      Coil( "E98" )
   END_RUNG
   // the same network as SCL:
   "E98" := "E6.0";
END_REGION

REGION Network 53: Top carriage up (Top)
   RUNG wire#powerrail
      Contact( "E6.1" )
      Coil( "E97" )
   END_RUNG
   // the same network as SCL:
   "E97" := "E6.1";
END_REGION

REGION Network 54: Reading pallet height for top carriage (Top)
   RUNG wire#powerrail
      Contact( "E6.2" )
      Coil( "E101" )
   END_RUNG
   // the same network as SCL:
   "E101" := "E6.2";
END_REGION

REGION Network 55: Clamp to block top film closed (Top)
   RUNG wire#powerrail
      Contact( "E6.3" )
      Coil( "E105" )
   END_RUNG
   // the same network as SCL:
   "E105" := "E6.3";
END_REGION

REGION Network 56: Top film cutter forward (Top)
   RUNG wire#powerrail
      Contact( "E6.4" )
      Coil( "E103" )
   END_RUNG
   // the same network as SCL:
   "E103" := "E6.4";
END_REGION

REGION Network 57: Top film cutter backward (Top)
   RUNG wire#powerrail
      Contact( "E6.5" )
      Coil( "E104" )
   END_RUNG
   // the same network as SCL:
   "E104" := "E6.5";
END_REGION

REGION Network 58: Top film ended sensor (Top)
   RUNG wire#powerrail
      Contact( "E6.6" )
      Coil( "E107" )
   END_RUNG
   // the same network as SCL:
   "E107" := "E6.6";
END_REGION

REGION Network 59: Top carriage position under pressure plate (Top)
   RUNG wire#powerrail
      Contact( "E110" )
      Coil( "E110" )
   END_RUNG
   // the same network as SCL:
   "E110" := "E110";
END_REGION

REGION Network 60: Top carriage backward (Top)
   RUNG wire#powerrail
      Contact( "E7.0" )
      Coil( "E99" )
   END_RUNG
   // the same network as SCL:
   "E99" := "E7.0";
END_REGION

REGION Network 61: Top carriage forward (Top)
   RUNG wire#powerrail
      Contact( "E7.1" )
      Coil( "E100" )
   END_RUNG
   // the same network as SCL:
   "E100" := "E7.1";
END_REGION

REGION Network 62: Clamp to pull top film closed (Top)
   RUNG wire#powerrail
      Contact( "E7.3" )
      Coil( "E106" )
   END_RUNG
   // the same network as SCL:
   "E106" := "E7.3";
END_REGION

REGION Network 63: Safety for top carriage movement (Top)
   RUNG wire#powerrail
      Contact( "E7.4" )
      Coil( "E102" )
   END_RUNG
   // the same network as SCL:
   "E102" := "E7.4";
END_REGION

REGION Network 64: Safety for top carriage downward for infeed conveyor (Top)
   RUNG wire#powerrail
      Contact( "E7.5" )
      Coil( "E108" )
   END_RUNG
   // the same network as SCL:
   "E108" := "E7.5";
END_REGION

REGION Network 65: Safety for top carriage downward for outfeed conveyor (Top)
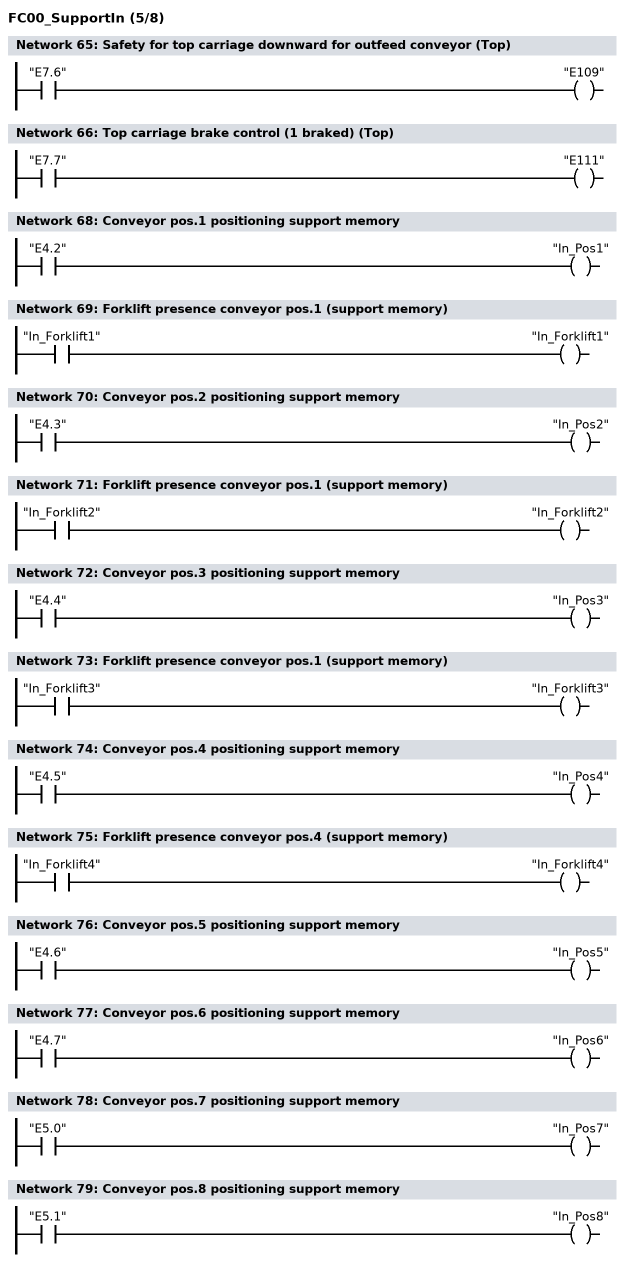
   RUNG wire#powerrail
      Contact( "E7.6" )
      Coil( "E109" )
   END_RUNG
   // the same network as SCL:
   "E109" := "E7.6";
END_REGION

REGION Network 66: Top carriage brake control (1 braked) (Top)
   RUNG wire#powerrail
      Contact( "E7.7" )
      Coil( "E111" )
   END_RUNG
   // the same network as SCL:
   "E111" := "E7.7";
END_REGION

REGION Network 67: ***CONVEYORS***
END_REGION

REGION Network 68: Conveyor pos.1 positioning support memory
   RUNG wire#powerrail
      Contact( "E4.2" )
      Coil( "In_Pos1" )
   END_RUNG
   // the same network as SCL:
   "In_Pos1" := "E4.2";
END_REGION

REGION Network 69: Forklift presence conveyor pos.1 (support memory)
   RUNG wire#powerrail
      Contact( "In_Forklift1" )
      Coil( "In_Forklift1" )
   END_RUNG
   // the same network as SCL:
   "In_Forklift1" := "In_Forklift1";
END_REGION

REGION Network 70: Conveyor pos.2 positioning support memory
   RUNG wire#powerrail
      Contact( "E4.3" )
      Coil( "In_Pos2" )
   END_RUNG
   // the same network as SCL:
   "In_Pos2" := "E4.3";
END_REGION

REGION Network 71: Forklift presence conveyor pos.1 (support memory)
   RUNG wire#powerrail
      Contact( "In_Forklift2" )
      Coil( "In_Forklift2" )
   END_RUNG
   // the same network as SCL:
   "In_Forklift2" := "In_Forklift2";
END_REGION

REGION Network 72: Conveyor pos.3 positioning support memory
   RUNG wire#powerrail
      Contact( "E4.4" )
      Coil( "In_Pos3" )
   END_RUNG
   // the same network as SCL:
   "In_Pos3" := "E4.4";
END_REGION

REGION Network 73: Forklift presence conveyor pos.1 (support memory)
   RUNG wire#powerrail
      Contact( "In_Forklift3" )
      Coil( "In_Forklift3" )
   END_RUNG
   // the same network as SCL:
   "In_Forklift3" := "In_Forklift3";
END_REGION

REGION Network 74: Conveyor pos.4 positioning support memory
   RUNG wire#powerrail
      Contact( "E4.5" )
      Coil( "In_Pos4" )
   END_RUNG
   // the same network as SCL:
   "In_Pos4" := "E4.5";
END_REGION

REGION Network 75: Forklift presence conveyor pos.4 (support memory)
   RUNG wire#powerrail
      Contact( "In_Forklift4" )
      Coil( "In_Forklift4" )
   END_RUNG
   // the same network as SCL:
   "In_Forklift4" := "In_Forklift4";
END_REGION

REGION Network 76: Conveyor pos.5 positioning support memory
   RUNG wire#powerrail
      Contact( "E4.6" )
      Coil( "In_Pos5" )
   END_RUNG
   // the same network as SCL:
   "In_Pos5" := "E4.6";
END_REGION

REGION Network 77: Conveyor pos.6 positioning support memory
   RUNG wire#powerrail
      Contact( "E4.7" )
      Coil( "In_Pos6" )
   END_RUNG
   // the same network as SCL:
   "In_Pos6" := "E4.7";
END_REGION

REGION Network 78: Conveyor pos.7 positioning support memory
   RUNG wire#powerrail
      Contact( "E5.0" )
      Coil( "In_Pos7" )
   END_RUNG
   // the same network as SCL:
   "In_Pos7" := "E5.0";
END_REGION

REGION Network 79: Conveyor pos.8 positioning support memory
   RUNG wire#powerrail
      Contact( "E5.1" )
      Coil( "In_Pos8" )
   END_RUNG
   // the same network as SCL:
   "In_Pos8" := "E5.1";
END_REGION

REGION Network 80: OTHER
END_REGION

REGION Network 81: Table rotation phase sensor (Technoplat)
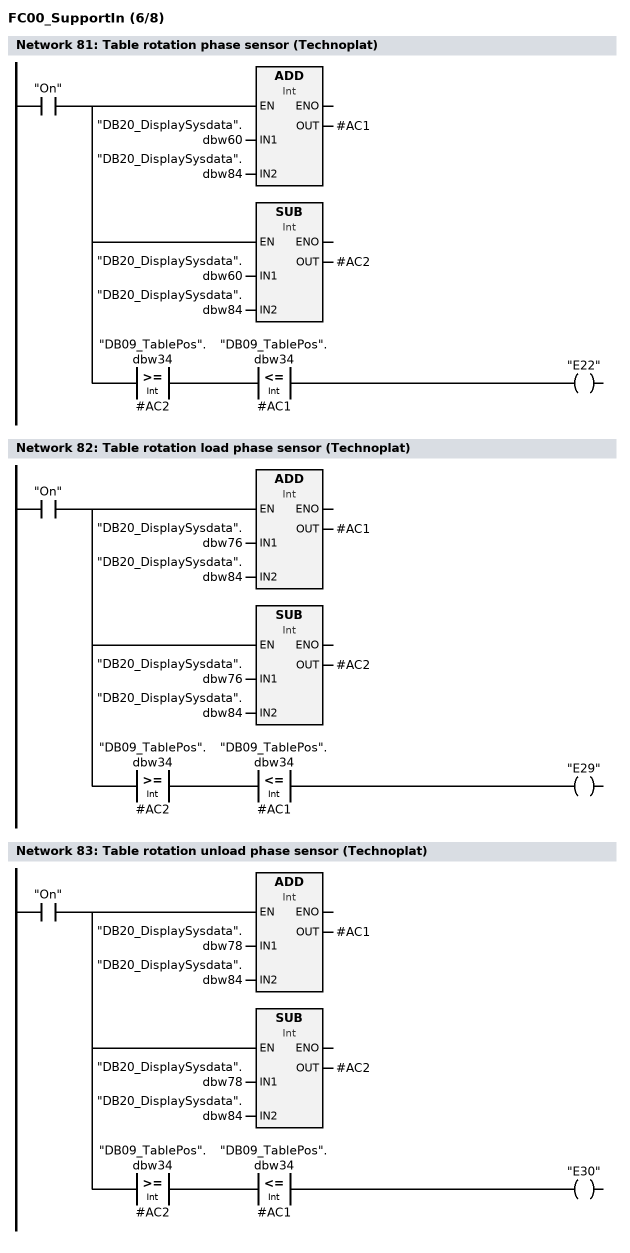
   RUNG wire#powerrail
      Contact( "On" )
      wire#w1
      { S7_Templates := "SrcType := Int"; S7_GenerateENO := "TRUE" } Add(in1 := "DB20_DisplaySysdata".dbw60, in2 := "DB20_DisplaySysdata".dbw84, out => #AC1)
   END_RUNG
   RUNG wire#w1
      { S7_Templates := "SrcType := Int"; S7_GenerateENO := "TRUE" } Sub(in1 := "DB20_DisplaySysdata".dbw60, in2 := "DB20_DisplaySysdata".dbw84, out => #AC2)
   END_RUNG
   RUNG wire#w1
      { S7_Templates := "SrcType := Int" } GE_Contact(in1 := "DB09_TablePos".dbw34, in2 := #AC2)
      { S7_Templates := "SrcType := Int" } LE_Contact(in1 := "DB09_TablePos".dbw34, in2 := #AC1)
      Coil( "E22" )
   END_RUNG
   // the same network as SCL:
   IF "On" THEN
       #AC1 := "DB20_DisplaySysdata".dbw60 + "DB20_DisplaySysdata".dbw84;
       #AC2 := "DB20_DisplaySysdata".dbw60 - "DB20_DisplaySysdata".dbw84;
   END_IF;
   "E22" := "On" AND ("DB09_TablePos".dbw34 >= #AC2) AND ("DB09_TablePos".dbw34 <= #AC1);
END_REGION

REGION Network 82: Table rotation load phase sensor (Technoplat)
   RUNG wire#powerrail
      Contact( "On" )
      wire#w1
      { S7_Templates := "SrcType := Int"; S7_GenerateENO := "TRUE" } Add(in1 := "DB20_DisplaySysdata".dbw76, in2 := "DB20_DisplaySysdata".dbw84, out => #AC1)
   END_RUNG
   RUNG wire#w1
      { S7_Templates := "SrcType := Int"; S7_GenerateENO := "TRUE" } Sub(in1 := "DB20_DisplaySysdata".dbw76, in2 := "DB20_DisplaySysdata".dbw84, out => #AC2)
   END_RUNG
   RUNG wire#w1
      { S7_Templates := "SrcType := Int" } GE_Contact(in1 := "DB09_TablePos".dbw34, in2 := #AC2)
      { S7_Templates := "SrcType := Int" } LE_Contact(in1 := "DB09_TablePos".dbw34, in2 := #AC1)
      Coil( "E29" )
   END_RUNG
   // the same network as SCL:
   IF "On" THEN
       #AC1 := "DB20_DisplaySysdata".dbw76 + "DB20_DisplaySysdata".dbw84;
       #AC2 := "DB20_DisplaySysdata".dbw76 - "DB20_DisplaySysdata".dbw84;
   END_IF;
   "E29" := "On" AND ("DB09_TablePos".dbw34 >= #AC2) AND ("DB09_TablePos".dbw34 <= #AC1);
END_REGION

REGION Network 83: Table rotation unload phase sensor (Technoplat)
   RUNG wire#powerrail
      Contact( "On" )
      wire#w1
      { S7_Templates := "SrcType := Int"; S7_GenerateENO := "TRUE" } Add(in1 := "DB20_DisplaySysdata".dbw78, in2 := "DB20_DisplaySysdata".dbw84, out => #AC1)
   END_RUNG
   RUNG wire#w1
      { S7_Templates := "SrcType := Int"; S7_GenerateENO := "TRUE" } Sub(in1 := "DB20_DisplaySysdata".dbw78, in2 := "DB20_DisplaySysdata".dbw84, out => #AC2)
   END_RUNG
   RUNG wire#w1
      { S7_Templates := "SrcType := Int" } GE_Contact(in1 := "DB09_TablePos".dbw34, in2 := #AC2)
      { S7_Templates := "SrcType := Int" } LE_Contact(in1 := "DB09_TablePos".dbw34, in2 := #AC1)
      Coil( "E30" )
   END_RUNG
   // the same network as SCL:
   IF "On" THEN
       #AC1 := "DB20_DisplaySysdata".dbw78 + "DB20_DisplaySysdata".dbw84;
       #AC2 := "DB20_DisplaySysdata".dbw78 - "DB20_DisplaySysdata".dbw84;
   END_IF;
   "E30" := "On" AND ("DB09_TablePos".dbw34 >= #AC2) AND ("DB09_TablePos".dbw34 <= #AC1);
END_REGION

REGION Network 84: Table rotation phase sensor (Technoplat)
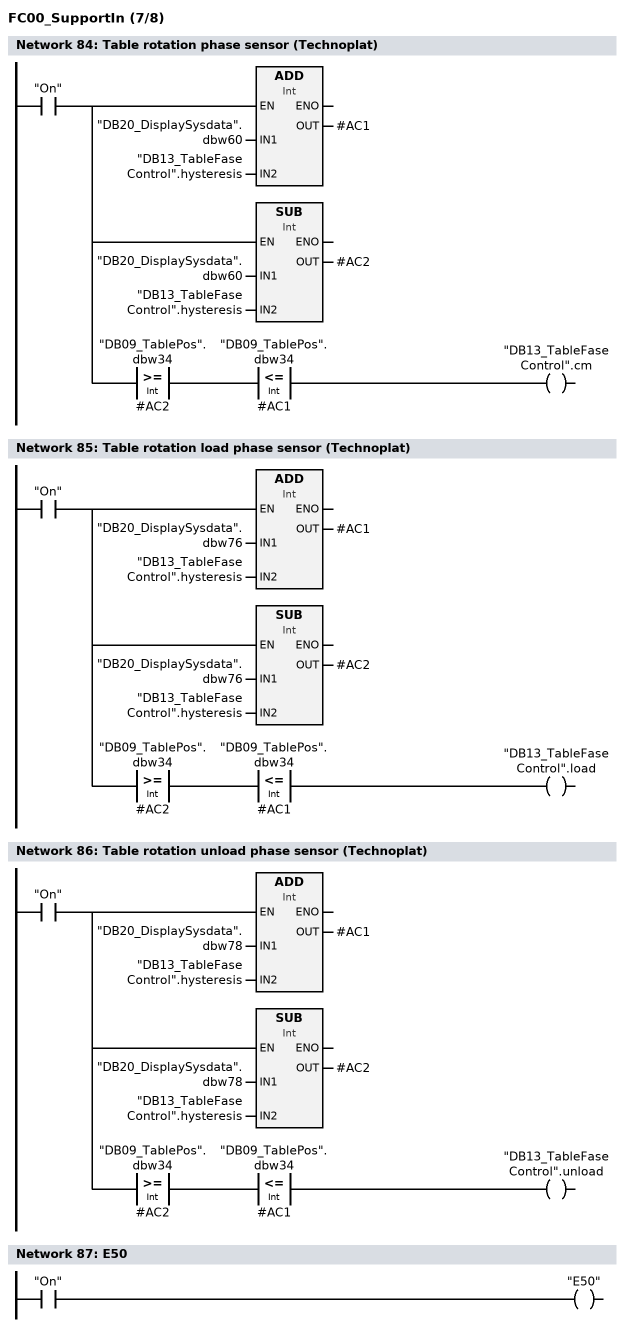
   RUNG wire#powerrail
      Contact( "On" )
      wire#w1
      { S7_Templates := "SrcType := Int"; S7_GenerateENO := "TRUE" } Add(in1 := "DB20_DisplaySysdata".dbw60, in2 := "DB13_TableFaseControl".hysteresis, out => #AC1)
   END_RUNG
   RUNG wire#w1
      { S7_Templates := "SrcType := Int"; S7_GenerateENO := "TRUE" } Sub(in1 := "DB20_DisplaySysdata".dbw60, in2 := "DB13_TableFaseControl".hysteresis, out => #AC2)
   END_RUNG
   RUNG wire#w1
      { S7_Templates := "SrcType := Int" } GE_Contact(in1 := "DB09_TablePos".dbw34, in2 := #AC2)
      { S7_Templates := "SrcType := Int" } LE_Contact(in1 := "DB09_TablePos".dbw34, in2 := #AC1)
      Coil( "DB13_TableFaseControl".cm )
   END_RUNG
   // the same network as SCL:
   IF "On" THEN
       #AC1 := "DB20_DisplaySysdata".dbw60 + "DB13_TableFaseControl".hysteresis;
       #AC2 := "DB20_DisplaySysdata".dbw60 - "DB13_TableFaseControl".hysteresis;
   END_IF;
   "DB13_TableFaseControl".cm := "On" AND ("DB09_TablePos".dbw34 >= #AC2) AND ("DB09_TablePos".dbw34 <= #AC1);
END_REGION

REGION Network 85: Table rotation load phase sensor (Technoplat)
   RUNG wire#powerrail
      Contact( "On" )
      wire#w1
      { S7_Templates := "SrcType := Int"; S7_GenerateENO := "TRUE" } Add(in1 := "DB20_DisplaySysdata".dbw76, in2 := "DB13_TableFaseControl".hysteresis, out => #AC1)
   END_RUNG
   RUNG wire#w1
      { S7_Templates := "SrcType := Int"; S7_GenerateENO := "TRUE" } Sub(in1 := "DB20_DisplaySysdata".dbw76, in2 := "DB13_TableFaseControl".hysteresis, out => #AC2)
   END_RUNG
   RUNG wire#w1
      { S7_Templates := "SrcType := Int" } GE_Contact(in1 := "DB09_TablePos".dbw34, in2 := #AC2)
      { S7_Templates := "SrcType := Int" } LE_Contact(in1 := "DB09_TablePos".dbw34, in2 := #AC1)
      Coil( "DB13_TableFaseControl".load )
   END_RUNG
   // the same network as SCL:
   IF "On" THEN
       #AC1 := "DB20_DisplaySysdata".dbw76 + "DB13_TableFaseControl".hysteresis;
       #AC2 := "DB20_DisplaySysdata".dbw76 - "DB13_TableFaseControl".hysteresis;
   END_IF;
   "DB13_TableFaseControl".load := "On" AND ("DB09_TablePos".dbw34 >= #AC2) AND ("DB09_TablePos".dbw34 <= #AC1);
END_REGION

REGION Network 86: Table rotation unload phase sensor (Technoplat)
   RUNG wire#powerrail
      Contact( "On" )
      wire#w1
      { S7_Templates := "SrcType := Int"; S7_GenerateENO := "TRUE" } Add(in1 := "DB20_DisplaySysdata".dbw78, in2 := "DB13_TableFaseControl".hysteresis, out => #AC1)
   END_RUNG
   RUNG wire#w1
      { S7_Templates := "SrcType := Int"; S7_GenerateENO := "TRUE" } Sub(in1 := "DB20_DisplaySysdata".dbw78, in2 := "DB13_TableFaseControl".hysteresis, out => #AC2)
   END_RUNG
   RUNG wire#w1
      { S7_Templates := "SrcType := Int" } GE_Contact(in1 := "DB09_TablePos".dbw34, in2 := #AC2)
      { S7_Templates := "SrcType := Int" } LE_Contact(in1 := "DB09_TablePos".dbw34, in2 := #AC1)
      Coil( "DB13_TableFaseControl".unload )
   END_RUNG
   // the same network as SCL:
   IF "On" THEN
       #AC1 := "DB20_DisplaySysdata".dbw78 + "DB13_TableFaseControl".hysteresis;
       #AC2 := "DB20_DisplaySysdata".dbw78 - "DB13_TableFaseControl".hysteresis;
   END_IF;
   "DB13_TableFaseControl".unload := "On" AND ("DB09_TablePos".dbw34 >= #AC2) AND ("DB09_TablePos".dbw34 <= #AC1);
END_REGION

REGION Network 87: E50
   RUNG wire#powerrail
      Contact( "On" )
      Coil( "E50" )
   END_RUNG
   // the same network as SCL:
   "E50" := "On";
END_REGION

REGION Network 88: OLD (NOT USED)
END_REGION

REGION Network 89: Key selector automatic (0)/manual (1) mode (Technoplat)
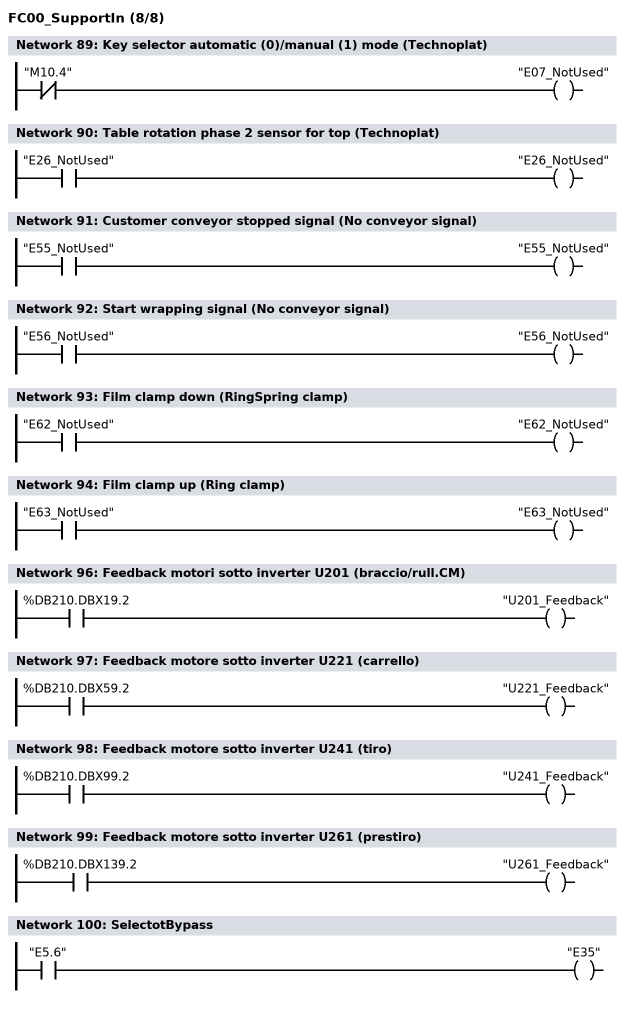
   RUNG wire#powerrail
      I_Contact( "M10.4" )
      Coil( "E07_NotUsed" )
   END_RUNG
   // the same network as SCL:
   "E07_NotUsed" := NOT "M10.4";
END_REGION

REGION Network 90: Table rotation phase 2 sensor for top (Technoplat)
   RUNG wire#powerrail
      Contact( "E26_NotUsed" )
      Coil( "E26_NotUsed" )
   END_RUNG
   // the same network as SCL:
   "E26_NotUsed" := "E26_NotUsed";
END_REGION

REGION Network 91: Customer conveyor stopped signal (No conveyor signal)
   RUNG wire#powerrail
      Contact( "E55_NotUsed" )
      Coil( "E55_NotUsed" )
   END_RUNG
   // the same network as SCL:
   "E55_NotUsed" := "E55_NotUsed";
END_REGION

REGION Network 92: Start wrapping signal (No conveyor signal)
   RUNG wire#powerrail
      Contact( "E56_NotUsed" )
      Coil( "E56_NotUsed" )
   END_RUNG
   // the same network as SCL:
   "E56_NotUsed" := "E56_NotUsed";
END_REGION

REGION Network 93: Film clamp down (RingSpring clamp)
   RUNG wire#powerrail
      Contact( "E62_NotUsed" )
      Coil( "E62_NotUsed" )
   END_RUNG
   // the same network as SCL:
   "E62_NotUsed" := "E62_NotUsed";
END_REGION

REGION Network 94: Film clamp up (Ring clamp)
   RUNG wire#powerrail
      Contact( "E63_NotUsed" )
      Coil( "E63_NotUsed" )
   END_RUNG
   // the same network as SCL:
   "E63_NotUsed" := "E63_NotUsed";
END_REGION

REGION Network 95: PROFINET DATA (inverter)
END_REGION

REGION Network 96: Feedback motori sotto inverter U201 (braccio/rull.CM)
   RUNG wire#powerrail
      Contact( %DB210.DBX19.2 )
      Coil( "U201_Feedback" )
   END_RUNG
   // the same network as SCL:
   "U201_Feedback" := %DB210.DBX19.2;
END_REGION

REGION Network 97: Feedback motore sotto inverter U221 (carrello)
   RUNG wire#powerrail
      Contact( %DB210.DBX59.2 )
      Coil( "U221_Feedback" )
   END_RUNG
   // the same network as SCL:
   "U221_Feedback" := %DB210.DBX59.2;
END_REGION

REGION Network 98: Feedback motore sotto inverter U241 (tiro)
   RUNG wire#powerrail
      Contact( %DB210.DBX99.2 )
      Coil( "U241_Feedback" )
   END_RUNG
   // the same network as SCL:
   "U241_Feedback" := %DB210.DBX99.2;
END_REGION

REGION Network 99: Feedback motore sotto inverter U261 (prestiro)
   RUNG wire#powerrail
      Contact( %DB210.DBX139.2 )
      Coil( "U261_Feedback" )
   END_RUNG
   // the same network as SCL:
   "U261_Feedback" := %DB210.DBX139.2;
END_REGION

REGION Network 100: SelectotBypass
   RUNG wire#powerrail
      Contact( "E5.6" )
      Coil( "E35" )
   END_RUNG
   // the same network as SCL:
   "E35" := "E5.6";
END_REGION
END_FUNCTION

FUNCTION "FC58_TableRotationPos" : Void   // FC58, LAD
{ S7_Optimized_Access := 'FALSE' }
VERSION : 0.1
// stored: AutoNumber false, IsIECCheckEnabled false, SetENOAutomatically false, UDAEnableTagReadback false
   VAR_INPUT
      PHASE : Bool;
   END_VAR
   VAR_TEMP
      TempDInt3 : DInt;
      PulseOffset : DInt;
      AC1 : Real;
      AC2 : Real;
      AC3 : Real;
      DeltaV : Real;
      DeltaVMax : Real;
      VattpiuVmin : Real;
      VmaxpiuVmin : Real;
      AC1_INT : Int;
      PulseReset : Bool;
      TEMPOMAX : Real;
      TEMPO : Real;
      Encoder : Int;
      TempDint : DInt;
      TempInt : Int;
      TempDint2 : DInt;
      TempDInt4 : DInt;
      TempWord : Word;
   END_VAR
   VAR_TEMP   // added for the SCL form of the ladder/FBD networks
      _w1 : Bool;
   END_VAR
BEGIN

REGION Network 1
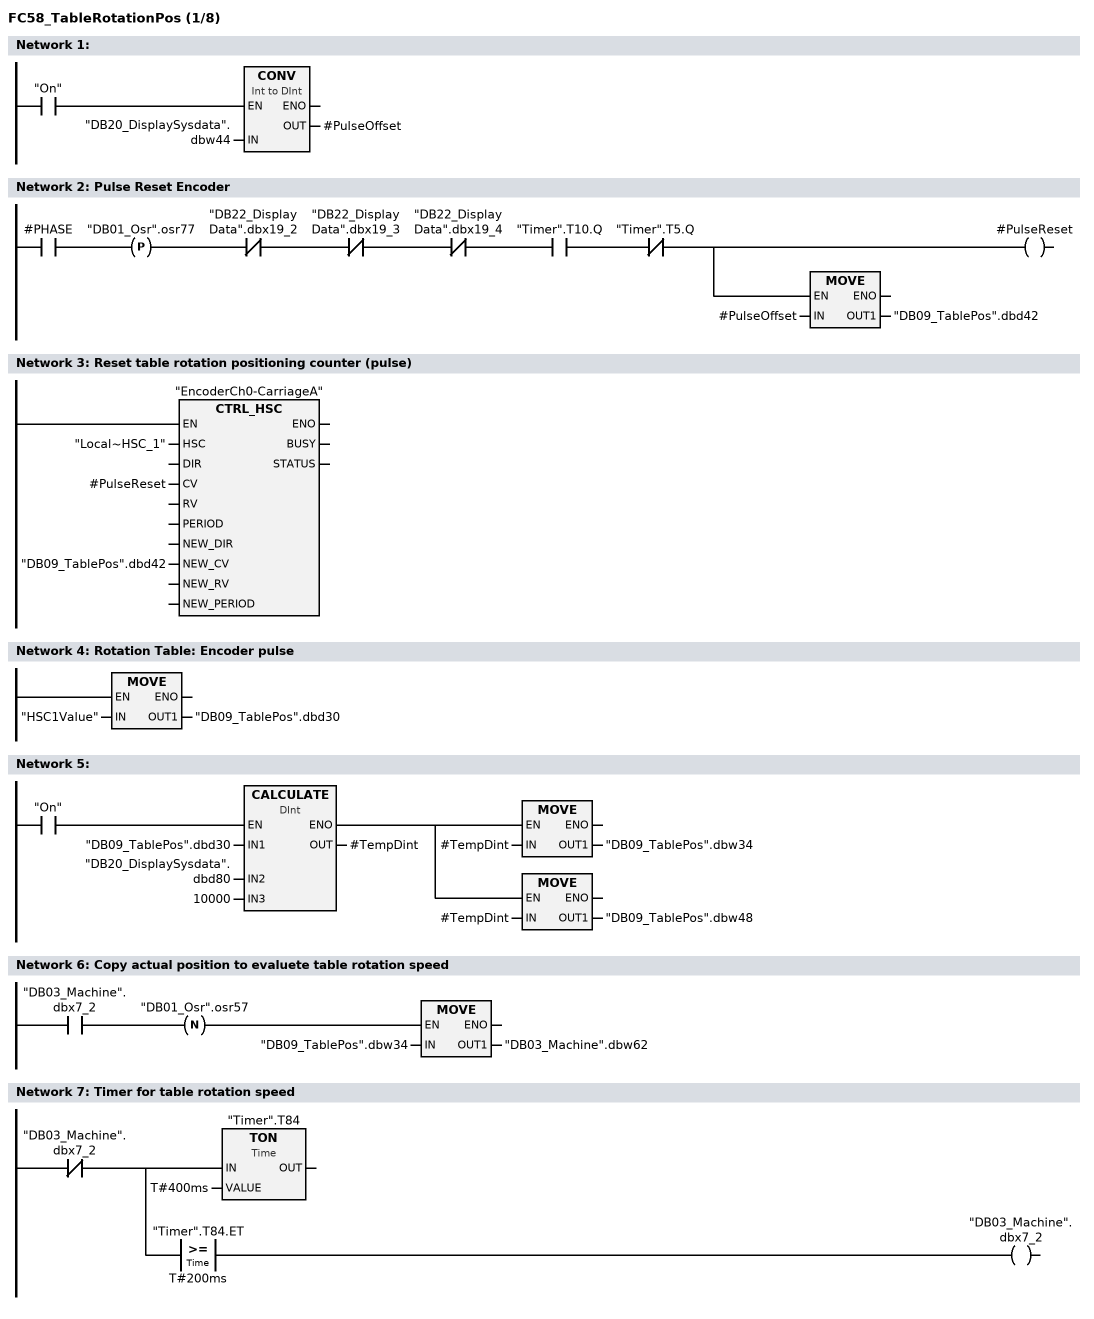
   RUNG wire#powerrail
      Contact( "On" )
      { S7_Templates := "[SrcType := Int, DestType := DInt]"; S7_GenerateENO := "TRUE" } Convert(in := "DB20_DisplaySysdata".dbw44, out => #PulseOffset)
   END_RUNG
   // the same network as SCL:
   IF "On" THEN #PulseOffset := INT_TO_DINT("DB20_DisplaySysdata".dbw44); END_IF;
END_REGION

REGION Network 2: Pulse Reset Encoder
   RUNG wire#powerrail
      Contact( #PHASE )
      P_Trig( "DB01_Osr".osr77 )
      I_Contact( "DB22_DisplayData".dbx19_2 )
      I_Contact( "DB22_DisplayData".dbx19_3 )
      I_Contact( "DB22_DisplayData".dbx19_4 )
      Contact( "Timer".T10.Q )
      I_Contact( "Timer".T5.Q )
      wire#w1
      Coil( #PulseReset )
   END_RUNG
   RUNG wire#w1
      { S7_GenerateENO := "TRUE" } Move(in := #PulseOffset, out1 => "DB09_TablePos".dbd42)
   END_RUNG
   // the same network as SCL:
   #_w1 := #PHASE AND NOT "DB01_Osr".osr77;   // rising edge
   "DB01_Osr".osr77 := #PHASE;
   #PulseReset := #_w1 AND NOT "DB22_DisplayData".dbx19_2 AND NOT "DB22_DisplayData".dbx19_3 AND NOT "DB22_DisplayData".dbx19_4 AND "Timer".T10.Q AND NOT "Timer".T5.Q;
   IF #PulseReset THEN "DB09_TablePos".dbd42 := #PulseOffset; END_IF;
END_REGION

REGION Network 3: Reset table rotation positioning counter (pulse)
   RUNG wire#powerrail
      "EncoderCh0-CarriageA".CTRL_HSC(HSC := "Local~HSC_1", DIR :=, CV := #PulseReset, RV :=, PERIOD :=, NEW_DIR :=, NEW_CV := "DB09_TablePos".dbd42, NEW_RV :=, NEW_PERIOD :=, BUSY =>, STATUS =>)
   END_RUNG
   // the same network as SCL:
   "EncoderCh0-CarriageA"(HSC := "Local~HSC_1", CV := #PulseReset, NEW_CV := "DB09_TablePos".dbd42);   // CTRL_HSC
END_REGION

REGION Network 4: Rotation Table: Encoder pulse
   RUNG wire#powerrail
      { S7_GenerateENO := "TRUE" } Move(in := "HSC1Value", out1 => "DB09_TablePos".dbd30)
   END_RUNG
   // the same network as SCL:
   "DB09_TablePos".dbd30 := "HSC1Value";
END_REGION

REGION Network 5
   RUNG wire#powerrail
      Contact( "On" )
      { S7_Templates := "SrcType := DInt"; S7_GenerateENO := "TRUE"; S7_Expression := "((In1*In2)/In3)" } Calculate(in1 := "DB09_TablePos".dbd30, in2 := "DB20_DisplaySysdata".dbd80, in3 := 10000, out => #TempDint)
      wire#w1
      { S7_GenerateENO := "TRUE" } Move(in := #TempDint, out1 => "DB09_TablePos".dbw34)
   END_RUNG
   RUNG wire#w1
      { S7_GenerateENO := "TRUE" } Move(in := #TempDint, out1 => "DB09_TablePos".dbw48)
   END_RUNG
   // the same network as SCL:
   // ENO of a box is taken as its EN; it also drops when the box reports an error
   IF "On" THEN
       #TempDint := (("DB09_TablePos".dbd30*"DB20_DisplaySysdata".dbd80)/10000);
       "DB09_TablePos".dbw34 := #TempDint;
       "DB09_TablePos".dbw48 := #TempDint;
   END_IF;
END_REGION

REGION Network 6: Copy actual position to evaluete table rotation speed
   RUNG wire#powerrail
      Contact( "DB03_Machine".dbx7_2 )
      N_Trig( "DB01_Osr".osr57 )
      { S7_GenerateENO := "TRUE" } Move(in := "DB09_TablePos".dbw34, out1 => "DB03_Machine".dbw62)
   END_RUNG
   // the same network as SCL:
   #_w1 := NOT "DB03_Machine".dbx7_2 AND "DB01_Osr".osr57;   // falling edge
   "DB01_Osr".osr57 := "DB03_Machine".dbx7_2;
   IF #_w1 THEN "DB03_Machine".dbw62 := "DB09_TablePos".dbw34; END_IF;
END_REGION

REGION Network 7: Timer for table rotation speed
   #_w1 := NOT "DB03_Machine".dbx7_2;
   "Timer".T84.TON(IN := #_w1, PT := T#400ms);   // TON coil
   "DB03_Machine".dbx7_2 := #_w1 AND ("Timer".T84.ET >= T#200ms);
END_REGION

REGION Network 8: Speed calculation (1)
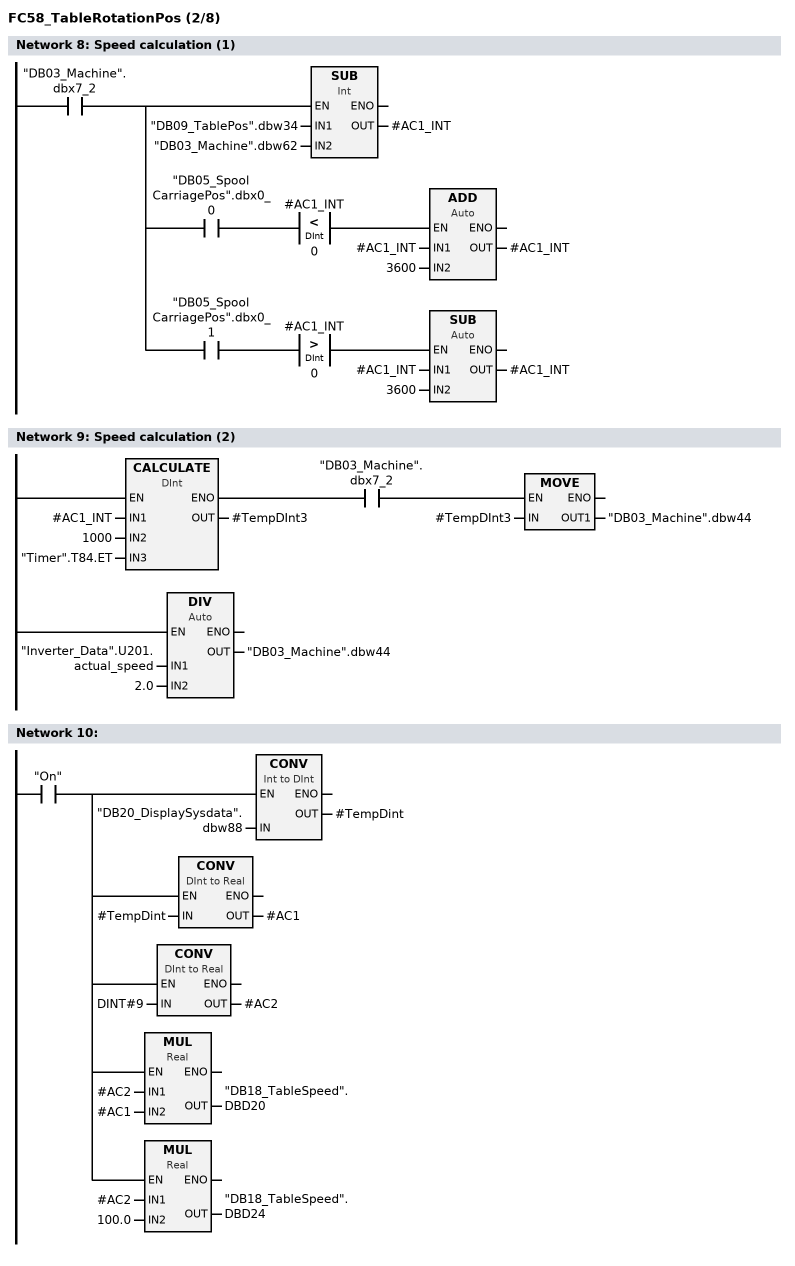
   RUNG wire#powerrail
      Contact( "DB03_Machine".dbx7_2 )
      wire#w1
      { S7_Templates := "SrcType := Int"; S7_GenerateENO := "TRUE" } Sub(in1 := "DB09_TablePos".dbw34, in2 := "DB03_Machine".dbw62, out => #AC1_INT)
   END_RUNG
   RUNG wire#w1
      Contact( "DB05_SpoolCarriagePos".dbx0_0 )
      { S7_Templates := "SrcType := DInt" } LT_Contact(in1 := #AC1_INT, in2 := 0)
      { S7_GenerateENO := "TRUE" } Add(in1 := #AC1_INT, in2 := 3600, out => #AC1_INT)
   END_RUNG
   RUNG wire#w1
      Contact( "DB05_SpoolCarriagePos".dbx0_1 )
      { S7_Templates := "SrcType := DInt" } GT_Contact(in1 := #AC1_INT, in2 := 0)
      { S7_GenerateENO := "TRUE" } Sub(in1 := #AC1_INT, in2 := 3600, out => #AC1_INT)
   END_RUNG
   // the same network as SCL:
   IF "DB03_Machine".dbx7_2 THEN #AC1_INT := "DB09_TablePos".dbw34 - "DB03_Machine".dbw62; END_IF;
   IF "DB03_Machine".dbx7_2 AND "DB05_SpoolCarriagePos".dbx0_0 AND (#AC1_INT < 0) THEN
       #AC1_INT := #AC1_INT + 3600;
   END_IF;
   IF "DB03_Machine".dbx7_2 AND "DB05_SpoolCarriagePos".dbx0_1 AND (#AC1_INT > 0) THEN
       #AC1_INT := #AC1_INT - 3600;
   END_IF;
END_REGION

REGION Network 9: Speed calculation (2)
   RUNG wire#powerrail
      { S7_Templates := "SrcType := DInt"; S7_GenerateENO := "TRUE"; S7_Expression := "((In1*In2)/In3)" } Calculate(in1 := #AC1_INT, in2 := 1000, in3 := "Timer".T84.ET, out => #TempDInt3)
      Contact( "DB03_Machine".dbx7_2 )
      { S7_GenerateENO := "TRUE" } Move(in := #TempDInt3, out1 => "DB03_Machine".dbw44)
   END_RUNG
   RUNG wire#powerrail
      Div(in1 := "Inverter_Data".U201.actual_speed, in2 := 2.0, out => "DB03_Machine".dbw44)
   END_RUNG
   // the same network as SCL:
   // ENO of a box is taken as its EN; it also drops when the box reports an error
   #TempDInt3 := ((#AC1_INT*1000)/"Timer".T84.ET);
   IF "DB03_Machine".dbx7_2 THEN "DB03_Machine".dbw44 := #TempDInt3; END_IF;
   "DB03_Machine".dbw44 := "Inverter_Data".U201.actual_speed / 2.0;
END_REGION

REGION Network 10
   RUNG wire#powerrail
      Contact( "On" )
      wire#w1
      { S7_Templates := "[SrcType := Int, DestType := DInt]"; S7_GenerateENO := "TRUE" } Convert(in := "DB20_DisplaySysdata".dbw88, out => #TempDint)
   END_RUNG
   RUNG wire#w1
      { S7_Templates := "[SrcType := DInt, DestType := Real]"; S7_GenerateENO := "TRUE" } Convert(in := #TempDint, out => #AC1)
   END_RUNG
   RUNG wire#w1
      { S7_Templates := "[SrcType := DInt, DestType := Real]"; S7_GenerateENO := "TRUE" } Convert(in := DINT#9, out => #AC2)
   END_RUNG
   RUNG wire#w1
      { S7_Templates := "SrcType := Real"; S7_GenerateENO := "TRUE" } Mul(in1 := #AC2, in2 := #AC1, out => "DB18_TableSpeed".DBD20)
   END_RUNG
   RUNG wire#w1
      { S7_Templates := "SrcType := Real"; S7_GenerateENO := "TRUE" } Mul(in1 := #AC2, in2 := 100.0, out => "DB18_TableSpeed".DBD24)
   END_RUNG
   // the same network as SCL:
   IF "On" THEN
       #TempDint := INT_TO_DINT("DB20_DisplaySysdata".dbw88);
       #AC1 := DINT_TO_REAL(#TempDint);
       #AC2 := DINT_TO_REAL(DINT#9);
       "DB18_TableSpeed".DBD20 := #AC2 * #AC1;
       "DB18_TableSpeed".DBD24 := #AC2 * 100.0;
   END_IF;
END_REGION

REGION Network 11
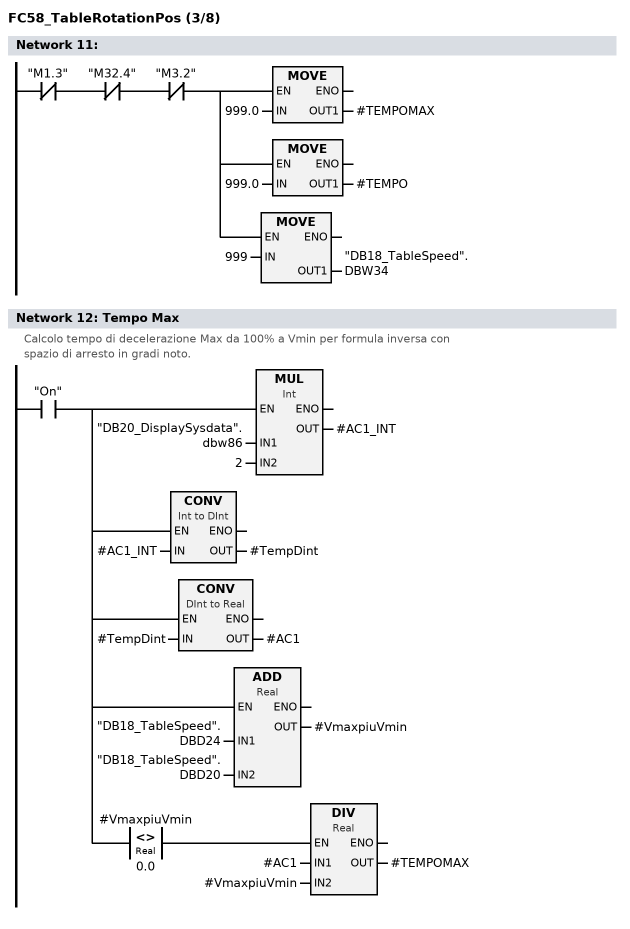
   RUNG wire#powerrail
      I_Contact( "M1.3" )
      I_Contact( "M32.4" )
      I_Contact( "M3.2" )
      wire#w1
      { S7_GenerateENO := "TRUE" } Move(in := 999.0, out1 => #TEMPOMAX)
   END_RUNG
   RUNG wire#w1
      { S7_GenerateENO := "TRUE" } Move(in := 999.0, out1 => #TEMPO)
   END_RUNG
   RUNG wire#w1
      { S7_GenerateENO := "TRUE" } Move(in := 999, out1 => "DB18_TableSpeed".DBW34)
   END_RUNG
   // the same network as SCL:
   IF NOT "M1.3" AND NOT "M32.4" AND NOT "M3.2" THEN
       #TEMPOMAX := 999.0;
       #TEMPO := 999.0;
       "DB18_TableSpeed".DBW34 := 999;
   END_IF;
END_REGION

REGION Network 12: Tempo Max
   // Calcolo tempo di decelerazione Max da 100% a Vmin per formula inversa con 
   // spazio di arresto in gradi noto.
   RUNG wire#powerrail
      Contact( "On" )
      wire#w1
      { S7_Templates := "SrcType := Int"; S7_GenerateENO := "TRUE" } Mul(in1 := "DB20_DisplaySysdata".dbw86, in2 := 2, out => #AC1_INT)
   END_RUNG
   RUNG wire#w1
      { S7_Templates := "[SrcType := Int, DestType := DInt]"; S7_GenerateENO := "TRUE" } Convert(in := #AC1_INT, out => #TempDint)
   END_RUNG
   RUNG wire#w1
      { S7_Templates := "[SrcType := DInt, DestType := Real]"; S7_GenerateENO := "TRUE" } Convert(in := #TempDint, out => #AC1)
   END_RUNG
   RUNG wire#w1
      { S7_Templates := "SrcType := Real"; S7_GenerateENO := "TRUE" } Add(in1 := "DB18_TableSpeed".DBD24, in2 := "DB18_TableSpeed".DBD20, out => #VmaxpiuVmin)
   END_RUNG
   RUNG wire#w1
      { S7_Templates := "SrcType := Real" } NE_Contact(in1 := #VmaxpiuVmin, in2 := 0.0)
      { S7_Templates := "SrcType := Real"; S7_GenerateENO := "TRUE" } Div(in1 := #AC1, in2 := #VmaxpiuVmin, out => #TEMPOMAX)
   END_RUNG
   // the same network as SCL:
   IF "On" THEN
       #AC1_INT := "DB20_DisplaySysdata".dbw86 * 2;
       #TempDint := INT_TO_DINT(#AC1_INT);
       #AC1 := DINT_TO_REAL(#TempDint);
       #VmaxpiuVmin := "DB18_TableSpeed".DBD24 + "DB18_TableSpeed".DBD20;
   END_IF;
   IF "On" AND (#VmaxpiuVmin <> 0.0) THEN #TEMPOMAX := #AC1 / #VmaxpiuVmin; END_IF;
END_REGION

REGION Network 13: Calcolo tempo di decelerazione da Vatt a Vmin per calcolo spazio di arresto
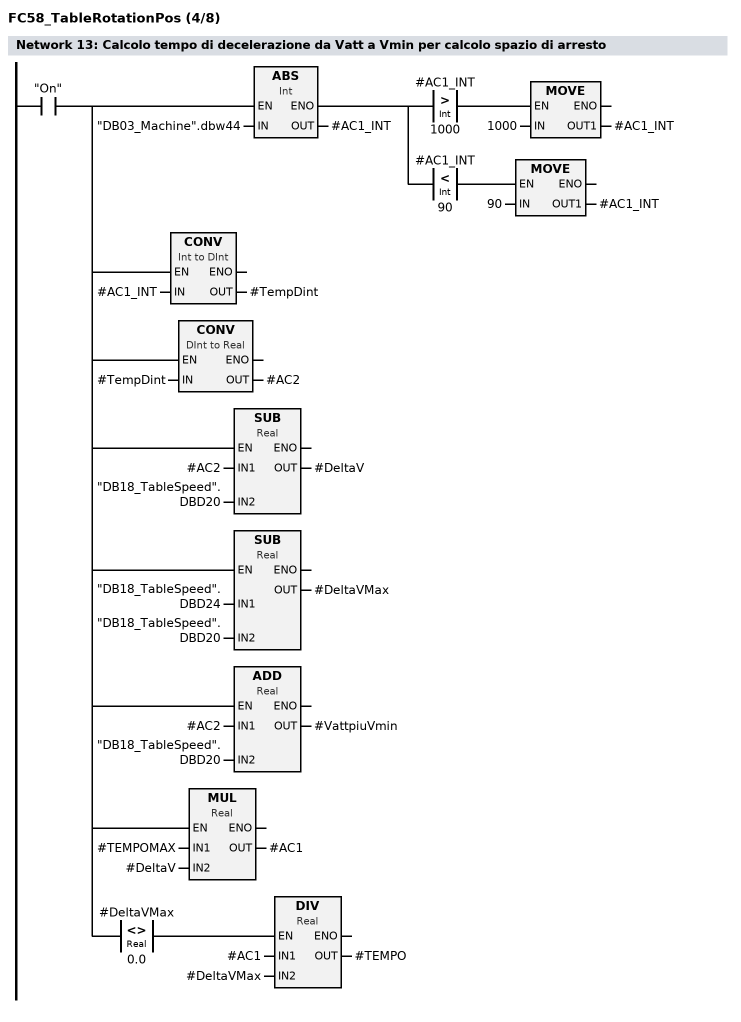
   RUNG wire#powerrail
      Contact( "On" )
      wire#w1
      { S7_Templates := "SrcType := Int" } Abs(in := "DB03_Machine".dbw44, out => #AC1_INT)
      wire#w2
      { S7_Templates := "SrcType := Int" } GT_Contact(in1 := #AC1_INT, in2 := 1000)
      Move(in := 1000, out1 => #AC1_INT)
   END_RUNG
   RUNG wire#w2
      { S7_Templates := "SrcType := Int" } LT_Contact(in1 := #AC1_INT, in2 := 90)
      Move(in := 90, out1 => #AC1_INT)
   END_RUNG
   RUNG wire#w1
      { S7_Templates := "[SrcType := Int, DestType := DInt]"; S7_GenerateENO := "TRUE" } Convert(in := #AC1_INT, out => #TempDint)
   END_RUNG
   RUNG wire#w1
      { S7_Templates := "[SrcType := DInt, DestType := Real]"; S7_GenerateENO := "TRUE" } Convert(in := #TempDint, out => #AC2)
   END_RUNG
   RUNG wire#w1
      { S7_Templates := "SrcType := Real"; S7_GenerateENO := "TRUE" } Sub(in1 := #AC2, in2 := "DB18_TableSpeed".DBD20, out => #DeltaV)
   END_RUNG
   RUNG wire#w1
      { S7_Templates := "SrcType := Real"; S7_GenerateENO := "TRUE" } Sub(in1 := "DB18_TableSpeed".DBD24, in2 := "DB18_TableSpeed".DBD20, out => #DeltaVMax)
   END_RUNG
   RUNG wire#w1
      { S7_Templates := "SrcType := Real"; S7_GenerateENO := "TRUE" } Add(in1 := #AC2, in2 := "DB18_TableSpeed".DBD20, out => #VattpiuVmin)
   END_RUNG
   RUNG wire#w1
      { S7_Templates := "SrcType := Real"; S7_GenerateENO := "TRUE" } Mul(in1 := #TEMPOMAX, in2 := #DeltaV, out => #AC1)
   END_RUNG
   RUNG wire#w1
      { S7_Templates := "SrcType := Real" } NE_Contact(in1 := #DeltaVMax, in2 := 0.0)
      { S7_Templates := "SrcType := Real"; S7_GenerateENO := "TRUE" } Div(in1 := #AC1, in2 := #DeltaVMax, out => #TEMPO)
   END_RUNG
   // the same network as SCL:
   IF "On" THEN #AC1_INT := ABS("DB03_Machine".dbw44); END_IF;
   IF "On" AND (#AC1_INT > 1000) THEN #AC1_INT := 1000; END_IF;
   IF "On" AND (#AC1_INT < 90) THEN #AC1_INT := 90; END_IF;
   IF "On" THEN
       #TempDint := INT_TO_DINT(#AC1_INT);
       #AC2 := DINT_TO_REAL(#TempDint);
       #DeltaV := #AC2 - "DB18_TableSpeed".DBD20;
       #DeltaVMax := "DB18_TableSpeed".DBD24 - "DB18_TableSpeed".DBD20;
       #VattpiuVmin := #AC2 + "DB18_TableSpeed".DBD20;
       #AC1 := #TEMPOMAX * #DeltaV;
   END_IF;
   IF "On" AND (#DeltaVMax <> 0.0) THEN #TEMPO := #AC1 / #DeltaVMax; END_IF;
END_REGION

REGION Network 14: Decelerazione
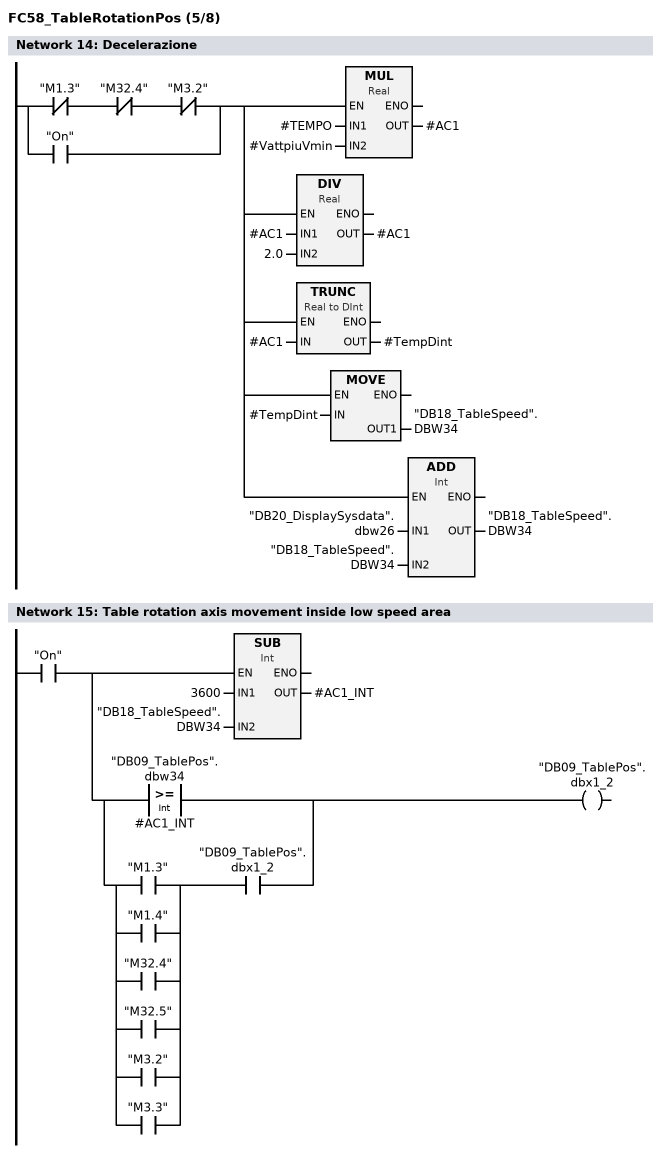
   RUNG wire#powerrail
      I_Contact( "M1.3" )
      I_Contact( "M32.4" )
      I_Contact( "M3.2" )
      wire#w1
      { S7_Templates := "SrcType := Real"; S7_GenerateENO := "TRUE" } Mul(in1 := #TEMPO, in2 := #VattpiuVmin, out => #AC1)
   END_RUNG
   RUNG wire#powerrail
      Contact( "On" )
   END_RUNG wire#w1
   RUNG wire#w1
      { S7_Templates := "SrcType := Real"; S7_GenerateENO := "TRUE" } Div(in1 := #AC1, in2 := 2.0, out => #AC1)
   END_RUNG
   RUNG wire#w1
      { S7_Templates := "[SrcType := Real, DestType := DInt]"; S7_GenerateENO := "TRUE" } Trunc(in := #AC1, out => #TempDint)
   END_RUNG
   RUNG wire#w1
      { S7_GenerateENO := "TRUE" } Move(in := #TempDint, out1 => "DB18_TableSpeed".DBW34)
   END_RUNG
   RUNG wire#w1
      { S7_Templates := "SrcType := Int"; S7_GenerateENO := "TRUE" } Add(in1 := "DB20_DisplaySysdata".dbw26, in2 := "DB18_TableSpeed".DBW34, out => "DB18_TableSpeed".DBW34)
   END_RUNG
   // the same network as SCL:
   IF (NOT "M1.3" AND NOT "M32.4" AND NOT "M3.2") OR "On" THEN
       #AC1 := #TEMPO * #VattpiuVmin;
       #AC1 := #AC1 / 2.0;
       #TempDint := TRUNC(#AC1);
       "DB18_TableSpeed".DBW34 := #TempDint;
       "DB18_TableSpeed".DBW34 := "DB20_DisplaySysdata".dbw26 + "DB18_TableSpeed".DBW34;
   END_IF;
END_REGION

REGION Network 15: Table rotation axis movement inside low speed area
   RUNG wire#powerrail
      Contact( "On" )
      wire#w1
      { S7_Templates := "SrcType := Int"; S7_GenerateENO := "TRUE" } Sub(in1 := 3600, in2 := "DB18_TableSpeed".DBW34, out => #AC1_INT)
   END_RUNG
   RUNG wire#w1
      { S7_Templates := "SrcType := Int" } GE_Contact(in1 := "DB09_TablePos".dbw34, in2 := #AC1_INT)
      wire#w2
      Coil( "DB09_TablePos".dbx1_2 )
   END_RUNG
   RUNG wire#w1
      Contact( "M1.3" )
      wire#w3
      Contact( "DB09_TablePos".dbx1_2 )
   END_RUNG wire#w2
   RUNG wire#w1
      Contact( "M1.4" )
   END_RUNG wire#w3
   RUNG wire#w1
      Contact( "M32.4" )
   END_RUNG wire#w3
   RUNG wire#w1
      Contact( "M32.5" )
   END_RUNG wire#w3
   RUNG wire#w1
      Contact( "M3.2" )
   END_RUNG wire#w3
   RUNG wire#w1
      Contact( "M3.3" )
   END_RUNG wire#w3
   // the same network as SCL:
   IF "On" THEN #AC1_INT := 3600 - "DB18_TableSpeed".DBW34; END_IF;
   "DB09_TablePos".dbx1_2 := "On" AND (("DB09_TablePos".dbw34 >= #AC1_INT) OR (("M1.3" OR "M1.4" OR "M32.4" OR "M32.5" OR "M3.2" OR "M3.3") AND "DB09_TablePos".dbx1_2));
END_REGION

REGION Network 16: Table rotation position loading/Unloading
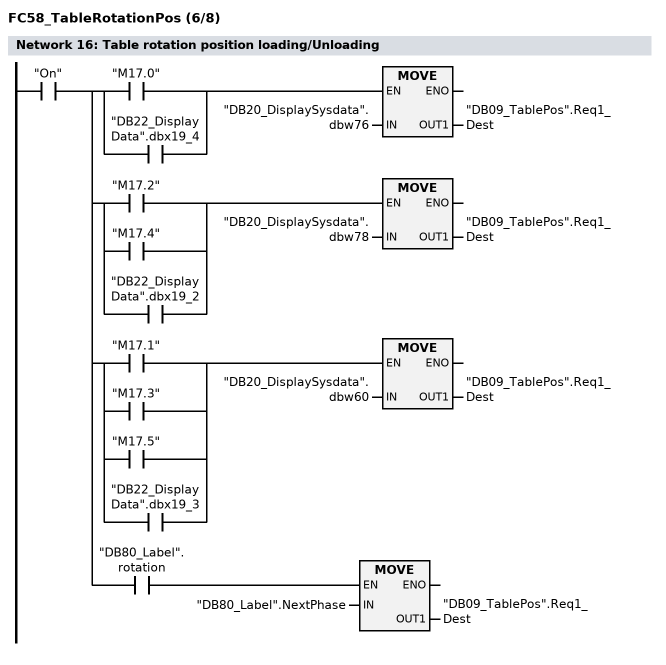
   RUNG wire#powerrail
      Contact( "On" )
      wire#w1
      Contact( "M17.0" )
      wire#w2
      { S7_GenerateENO := "TRUE" } Move(in := "DB20_DisplaySysdata".dbw76, out1 => "DB09_TablePos".Req1_Dest)
   END_RUNG
   RUNG wire#w1
      Contact( "DB22_DisplayData".dbx19_4 )
   END_RUNG wire#w2
   RUNG wire#w1
      Contact( "M17.2" )
      wire#w3
      { S7_GenerateENO := "TRUE" } Move(in := "DB20_DisplaySysdata".dbw78, out1 => "DB09_TablePos".Req1_Dest)
   END_RUNG
   RUNG wire#w1
      Contact( "M17.4" )
   END_RUNG wire#w3
   RUNG wire#w1
      Contact( "DB22_DisplayData".dbx19_2 )
   END_RUNG wire#w3
   RUNG wire#w1
      Contact( "M17.1" )
      wire#w4
      { S7_GenerateENO := "TRUE" } Move(in := "DB20_DisplaySysdata".dbw60, out1 => "DB09_TablePos".Req1_Dest)
   END_RUNG
   RUNG wire#w1
      Contact( "M17.3" )
   END_RUNG wire#w4
   RUNG wire#w1
      Contact( "M17.5" )
   END_RUNG wire#w4
   RUNG wire#w1
      Contact( "DB22_DisplayData".dbx19_3 )
   END_RUNG wire#w4
   RUNG wire#w1
      Contact( "DB80_Label".rotation )
      { S7_GenerateENO := "TRUE" } Move(in := "DB80_Label".NextPhase, out1 => "DB09_TablePos".Req1_Dest)
   END_RUNG
   // the same network as SCL:
   IF "On" AND ("M17.0" OR "DB22_DisplayData".dbx19_4) THEN
       "DB09_TablePos".Req1_Dest := "DB20_DisplaySysdata".dbw76;
   END_IF;
   IF "On" AND ("M17.2" OR "M17.4" OR "DB22_DisplayData".dbx19_2) THEN
       "DB09_TablePos".Req1_Dest := "DB20_DisplaySysdata".dbw78;
   END_IF;
   IF "On" AND ("M17.1" OR "M17.3" OR "M17.5" OR "DB22_DisplayData".dbx19_3) THEN
       "DB09_TablePos".Req1_Dest := "DB20_DisplaySysdata".dbw60;
   END_IF;
   IF "On" AND "DB80_Label".rotation THEN "DB09_TablePos".Req1_Dest := "DB80_Label".NextPhase; END_IF;
END_REGION

REGION Network 17
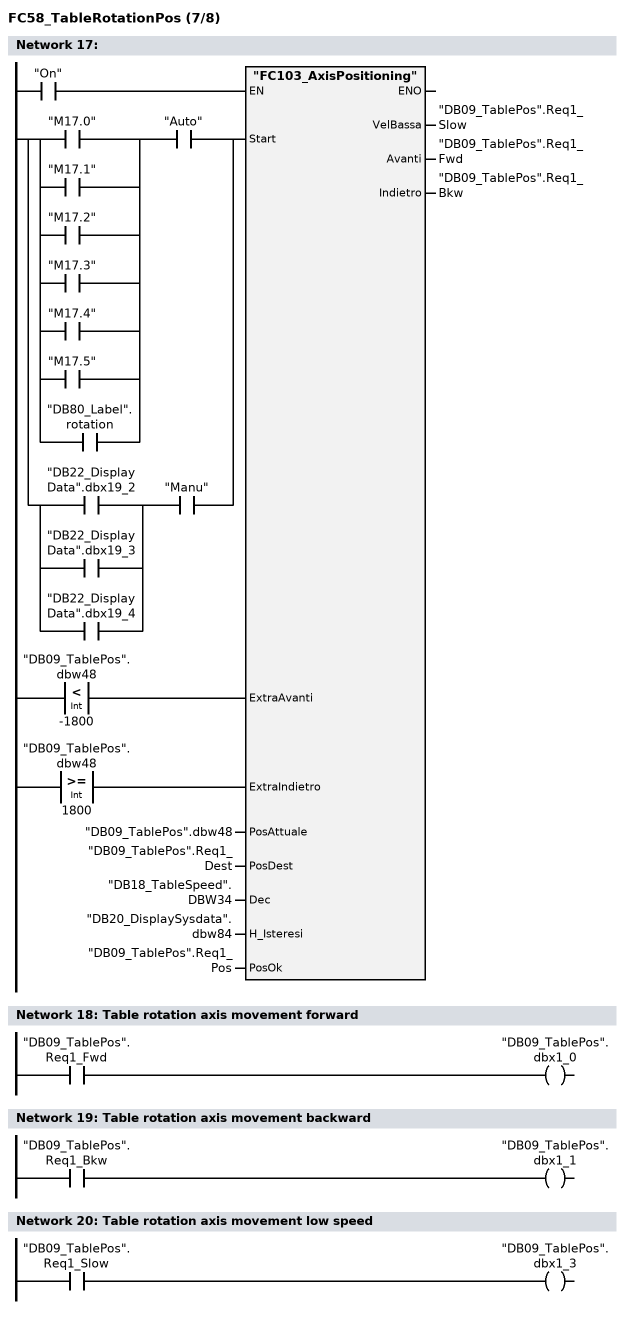
   RUNG wire#powerrail
      Contact( "On" )
      "FC103_AxisPositioning"(Start := wire#w3, ExtraAvanti := wire#w4, ExtraIndietro := wire#w5, PosAttuale := "DB09_TablePos".dbw48, PosDest := "DB09_TablePos".Req1_Dest, Dec := "DB18_TableSpeed".DBW34, H_Isteresi := "DB20_DisplaySysdata".dbw84, PosOk := "DB09_TablePos".Req1_Pos, VelBassa => "DB09_TablePos".Req1_Slow, Avanti => "DB09_TablePos".Req1_Fwd, Indietro => "DB09_TablePos".Req1_Bkw)
   END_RUNG
   RUNG wire#powerrail
      Contact( "M17.0" )
      wire#w1
      Contact( "Auto" )
   END_RUNG wire#w3
   RUNG wire#powerrail
      Contact( "M17.1" )
   END_RUNG wire#w1
   RUNG wire#powerrail
      Contact( "M17.2" )
   END_RUNG wire#w1
   RUNG wire#powerrail
      Contact( "M17.3" )
   END_RUNG wire#w1
   RUNG wire#powerrail
      Contact( "M17.4" )
   END_RUNG wire#w1
   RUNG wire#powerrail
      Contact( "M17.5" )
   END_RUNG wire#w1
   RUNG wire#powerrail
      Contact( "DB80_Label".rotation )
   END_RUNG wire#w1
   RUNG wire#powerrail
      Contact( "DB22_DisplayData".dbx19_2 )
      wire#w2
      Contact( "Manu" )
   END_RUNG wire#w3
   RUNG wire#powerrail
      Contact( "DB22_DisplayData".dbx19_3 )
   END_RUNG wire#w2
   RUNG wire#powerrail
      Contact( "DB22_DisplayData".dbx19_4 )
   END_RUNG wire#w2
   RUNG wire#powerrail
      { S7_Templates := "SrcType := Int" } LT_Contact(in1 := "DB09_TablePos".dbw48, in2 := -1800)
   END_RUNG wire#w4
   RUNG wire#powerrail
      { S7_Templates := "SrcType := Int" } GE_Contact(in1 := "DB09_TablePos".dbw48, in2 := 1800)
   END_RUNG wire#w5
   // the same network as SCL:
   IF "On" THEN
       "FC103_AxisPositioning"(Start := (("M17.0" OR "M17.1" OR "M17.2" OR "M17.3" OR "M17.4" OR "M17.5" OR "DB80_Label".rotation) AND "Auto") OR (("DB22_DisplayData".dbx19_2 OR "DB22_DisplayData".dbx19_3 OR "DB22_DisplayData".dbx19_4) AND "Manu"),
                               ExtraAvanti := "DB09_TablePos".dbw48 < (-1800),
                               ExtraIndietro := "DB09_TablePos".dbw48 >= 1800,
                               PosAttuale := "DB09_TablePos".dbw48,
                               PosDest := "DB09_TablePos".Req1_Dest,
                               Dec := "DB18_TableSpeed".DBW34,
                               H_Isteresi := "DB20_DisplaySysdata".dbw84,
                               PosOk := "DB09_TablePos".Req1_Pos,
                               VelBassa => "DB09_TablePos".Req1_Slow,
                               Avanti => "DB09_TablePos".Req1_Fwd,
                               Indietro => "DB09_TablePos".Req1_Bkw);
   END_IF;
END_REGION

REGION Network 18: Table rotation axis movement forward
   RUNG wire#powerrail
      Contact( "DB09_TablePos".Req1_Fwd )
      Coil( "DB09_TablePos".dbx1_0 )
   END_RUNG
   // the same network as SCL:
   "DB09_TablePos".dbx1_0 := "DB09_TablePos".Req1_Fwd;
END_REGION

REGION Network 19: Table rotation axis movement backward
   RUNG wire#powerrail
      Contact( "DB09_TablePos".Req1_Bkw )
      Coil( "DB09_TablePos".dbx1_1 )
   END_RUNG
   // the same network as SCL:
   "DB09_TablePos".dbx1_1 := "DB09_TablePos".Req1_Bkw;
END_REGION

REGION Network 20: Table rotation axis movement low speed
   RUNG wire#powerrail
      Contact( "DB09_TablePos".Req1_Slow )
      Coil( "DB09_TablePos".dbx1_3 )
   END_RUNG
   // the same network as SCL:
   "DB09_TablePos".dbx1_3 := "DB09_TablePos".Req1_Slow;
END_REGION

REGION Network 21: TABLE ENCODER CHECK
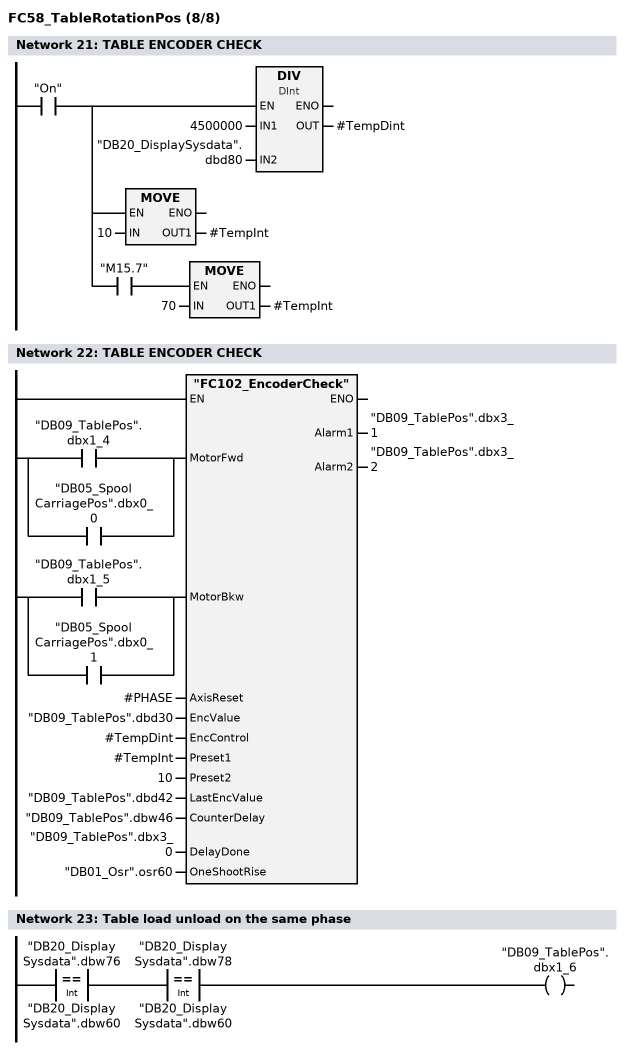
   RUNG wire#powerrail
      Contact( "On" )
      wire#w1
      { S7_Templates := "SrcType := DInt"; S7_GenerateENO := "TRUE" } Div(in1 := 4500000, in2 := "DB20_DisplaySysdata".dbd80, out => #TempDint)
   END_RUNG
   RUNG wire#w1
      { S7_GenerateENO := "TRUE" } Move(in := 10, out1 => #TempInt)
   END_RUNG
   RUNG wire#w1
      Contact( "M15.7" )
      { S7_GenerateENO := "TRUE" } Move(in := 70, out1 => #TempInt)
   END_RUNG
   // the same network as SCL:
   IF "On" THEN
       #TempDint := 4500000 / "DB20_DisplaySysdata".dbd80;
       #TempInt := 10;
   END_IF;
   IF "On" AND "M15.7" THEN #TempInt := 70; END_IF;
END_REGION

REGION Network 22: TABLE ENCODER CHECK
   RUNG wire#powerrail
      "FC102_EncoderCheck"(MotorFwd := wire#w1, MotorBkw := wire#w2, AxisReset := #PHASE, EncValue := "DB09_TablePos".dbd30, EncControl := #TempDint, Preset1 := #TempInt, Preset2 := 10, LastEncValue := "DB09_TablePos".dbd42, CounterDelay := "DB09_TablePos".dbw46, DelayDone := "DB09_TablePos".dbx3_0, OneShootRise := "DB01_Osr".osr60, Alarm1 => "DB09_TablePos".dbx3_1, Alarm2 => "DB09_TablePos".dbx3_2)
   END_RUNG
   RUNG wire#powerrail
      Contact( "DB09_TablePos".dbx1_4 )
   END_RUNG wire#w1
   RUNG wire#powerrail
      Contact( "DB05_SpoolCarriagePos".dbx0_0 )
   END_RUNG wire#w1
   RUNG wire#powerrail
      Contact( "DB09_TablePos".dbx1_5 )
   END_RUNG wire#w2
   RUNG wire#powerrail
      Contact( "DB05_SpoolCarriagePos".dbx0_1 )
   END_RUNG wire#w2
   // the same network as SCL:
   "FC102_EncoderCheck"(MotorFwd := "DB09_TablePos".dbx1_4 OR "DB05_SpoolCarriagePos".dbx0_0,
                        MotorBkw := "DB09_TablePos".dbx1_5 OR "DB05_SpoolCarriagePos".dbx0_1,
                        AxisReset := #PHASE,
                        EncValue := "DB09_TablePos".dbd30,
                        EncControl := #TempDint,
                        Preset1 := #TempInt,
                        Preset2 := 10,
                        LastEncValue := "DB09_TablePos".dbd42,
                        CounterDelay := "DB09_TablePos".dbw46,
                        DelayDone := "DB09_TablePos".dbx3_0,
                        OneShootRise := "DB01_Osr".osr60,
                        Alarm1 => "DB09_TablePos".dbx3_1,
                        Alarm2 => "DB09_TablePos".dbx3_2);
END_REGION

REGION Network 23: Table load unload on the same phase
   RUNG wire#powerrail
      { S7_Templates := "SrcType := Int" } EQ_Contact(in1 := "DB20_DisplaySysdata".dbw76, in2 := "DB20_DisplaySysdata".dbw60)
      { S7_Templates := "SrcType := Int" } EQ_Contact(in1 := "DB20_DisplaySysdata".dbw78, in2 := "DB20_DisplaySysdata".dbw60)
      Coil( "DB09_TablePos".dbx1_6 )
   END_RUNG
   // the same network as SCL:
   "DB09_TablePos".dbx1_6 := ("DB20_DisplaySysdata".dbw76 = "DB20_DisplaySysdata".dbw60) AND ("DB20_DisplaySysdata".dbw78 = "DB20_DisplaySysdata".dbw60);
END_REGION
END_FUNCTION

FUNCTION "FC103_AxisPositioning" : Void   // FC103, LAD
TITLE = Axis positioning
{ S7_Optimized_Access := 'FALSE' }
AUTHOR : Robopac
VERSION : 0.0
// stored: AutoNumber false, IsIECCheckEnabled false, SetENOAutomatically false, UDAEnableTagReadback false
   VAR_INPUT
      Start : Bool;   // Start dell'asse
      ExtraAvanti : Bool;   // Sensore di extracorsa avanti
      ExtraIndietro : Bool;   // Sensore di extracorsa indietro
      PosAttuale : Int;   // Posizione attule dell'asse
      PosDest : Int;   // Posizione di destinazione dell'asse
      Dec : Int;   // Decelerazione
      H_Isteresi : Int;   // Isteresi
   END_VAR
   VAR_OUTPUT
      VelBassa : Bool;   // Asse all'interno dell'intervallo di decelerazione
      Avanti : Bool;   // Asse avanti
      Indietro : Bool;   // Asse indietro
   END_VAR
   VAR_IN_OUT
      PosOk : Bool;   // Asse in posizione
   END_VAR
   VAR_TEMP
      PosDestMenoH : Int;   // Posizione di destinazione asse-Isteresi
      PosDestPiuH : Int;   // Posizione di destinazione asse+Isteresi
      PosDestMenoDec : Int;   // Posizione di destinazione asse-Decelerazione
      PosDestPiuDec : Int;   // Posizione di destinazione asse+Decelerazione
   END_VAR
   VAR_TEMP   // added for the SCL form of the ladder/FBD networks
      _w1 : Bool;
   END_VAR
BEGIN

REGION Network 1
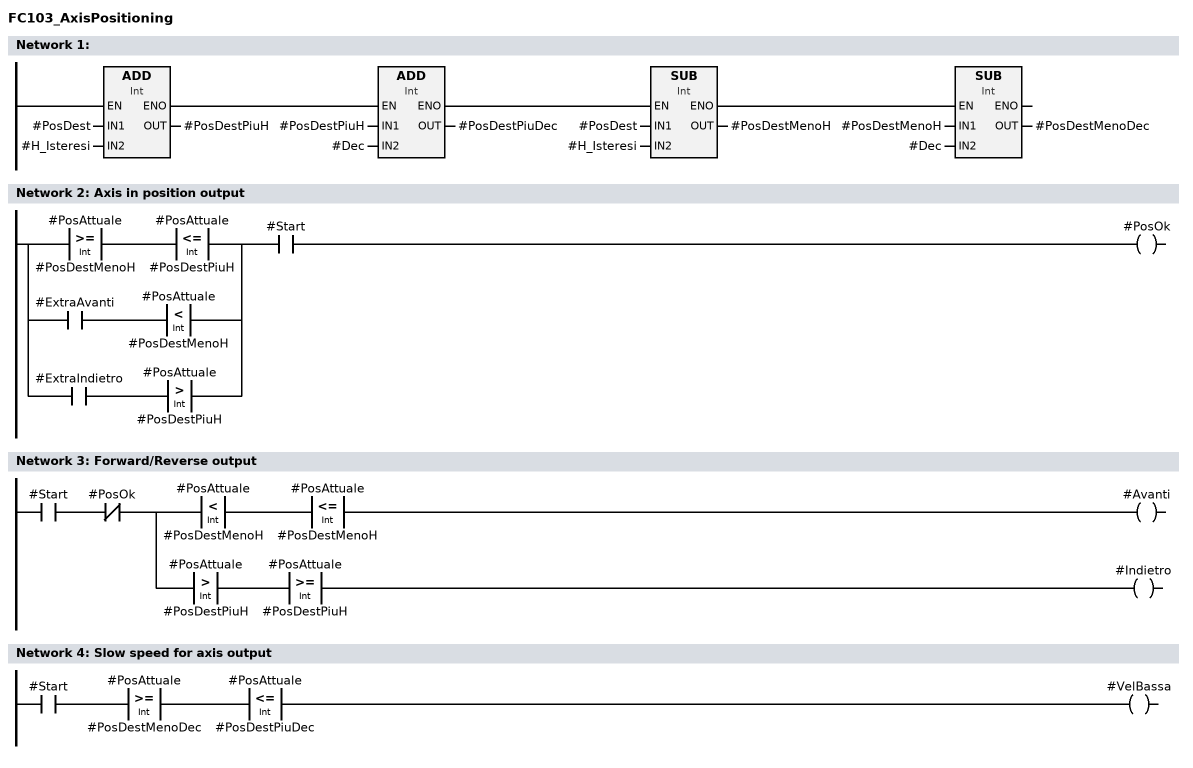
   RUNG wire#powerrail
      { S7_Templates := "SrcType := Int"; S7_GenerateENO := "TRUE" } Add(in1 := #PosDest, in2 := #H_Isteresi, out => #PosDestPiuH)
      { S7_Templates := "SrcType := Int"; S7_GenerateENO := "TRUE" } Add(in1 := #PosDestPiuH, in2 := #Dec, out => #PosDestPiuDec)
      { S7_Templates := "SrcType := Int"; S7_GenerateENO := "TRUE" } Sub(in1 := #PosDest, in2 := #H_Isteresi, out => #PosDestMenoH)
      { S7_Templates := "SrcType := Int"; S7_GenerateENO := "TRUE" } Sub(in1 := #PosDestMenoH, in2 := #Dec, out => #PosDestMenoDec)
   END_RUNG
   // the same network as SCL:
   // ENO of a box is taken as its EN; it also drops when the box reports an error
   #PosDestPiuH := #PosDest + #H_Isteresi;
   #PosDestPiuDec := #PosDestPiuH + #Dec;
   #PosDestMenoH := #PosDest - #H_Isteresi;
   #PosDestMenoDec := #PosDestMenoH - #Dec;
END_REGION

REGION Network 2: Axis in position output
   RUNG wire#powerrail
      { S7_Templates := "SrcType := Int" } GE_Contact(in1 := #PosAttuale, in2 := #PosDestMenoH)
      { S7_Templates := "SrcType := Int" } LE_Contact(in1 := #PosAttuale, in2 := #PosDestPiuH)
      wire#w1
      Contact( #Start )
      Coil( #PosOk )
   END_RUNG
   RUNG wire#powerrail
      Contact( #ExtraAvanti )
      { S7_Templates := "SrcType := Int" } LT_Contact(in1 := #PosAttuale, in2 := #PosDestMenoH)
   END_RUNG wire#w1
   RUNG wire#powerrail
      Contact( #ExtraIndietro )
      { S7_Templates := "SrcType := Int" } GT_Contact(in1 := #PosAttuale, in2 := #PosDestPiuH)
   END_RUNG wire#w1
   // the same network as SCL:
   #PosOk := (((#PosAttuale >= #PosDestMenoH) AND (#PosAttuale <= #PosDestPiuH)) OR (#ExtraAvanti AND (#PosAttuale < #PosDestMenoH)) OR (#ExtraIndietro AND (#PosAttuale > #PosDestPiuH))) AND #Start;
END_REGION

REGION Network 3: Forward/Reverse output
   RUNG wire#powerrail
      Contact( #Start )
      I_Contact( #PosOk )
      wire#w1
      { S7_Templates := "SrcType := Int" } LT_Contact(in1 := #PosAttuale, in2 := #PosDestMenoH)
      { S7_Templates := "SrcType := Int" } LE_Contact(in1 := #PosAttuale, in2 := #PosDestMenoH)
      Coil( #Avanti )
   END_RUNG
   RUNG wire#w1
      { S7_Templates := "SrcType := Int" } GT_Contact(in1 := #PosAttuale, in2 := #PosDestPiuH)
      { S7_Templates := "SrcType := Int" } GE_Contact(in1 := #PosAttuale, in2 := #PosDestPiuH)
      Coil( #Indietro )
   END_RUNG
   // the same network as SCL:
   #_w1 := #Start AND NOT #PosOk;
   #Avanti := #_w1 AND (#PosAttuale < #PosDestMenoH) AND (#PosAttuale <= #PosDestMenoH);
   #Indietro := #_w1 AND (#PosAttuale > #PosDestPiuH) AND (#PosAttuale >= #PosDestPiuH);
END_REGION

REGION Network 4: Slow speed for axis output
   RUNG wire#powerrail
      Contact( #Start )
      { S7_Templates := "SrcType := Int" } GE_Contact(in1 := #PosAttuale, in2 := #PosDestMenoDec)
      { S7_Templates := "SrcType := Int" } LE_Contact(in1 := #PosAttuale, in2 := #PosDestPiuDec)
      Coil( #VelBassa )
   END_RUNG
   // the same network as SCL:
   #VelBassa := #Start AND (#PosAttuale >= #PosDestMenoDec) AND (#PosAttuale <= #PosDestPiuDec);
END_REGION
END_FUNCTION

FUNCTION "FC102_EncoderCheck" : Void   // FC102, LAD
{ S7_Optimized_Access := 'FALSE' }
AUTHOR : AetnaG
VERSION : 0.0
// stored: AutoNumber false, IsIECCheckEnabled false, SetENOAutomatically false, UDAEnableTagReadback false
   VAR_INPUT
      MotorFwd : Bool;
      MotorBkw : Bool;
      AxisReset : Bool;
      EncValue : DInt;
      EncControl : DInt;
      Preset1 : Int;
      Preset2 : Int;
   END_VAR
   VAR_OUTPUT
      Alarm1 : Bool;
      Alarm2 : Bool;
   END_VAR
   VAR_IN_OUT
      LastEncValue : DInt;
      CounterDelay : Int;
      DelayDone : Bool;
      OneShootRise : Bool;
   END_VAR
   VAR_TEMP
      EncDifference : DInt;
      EncControlOpp : DInt;
      CounterReset : Bool;
   END_VAR
   VAR_TEMP   // added for the SCL form of the ladder/FBD networks
      _w1 : Bool;
   END_VAR
BEGIN

REGION Network 1
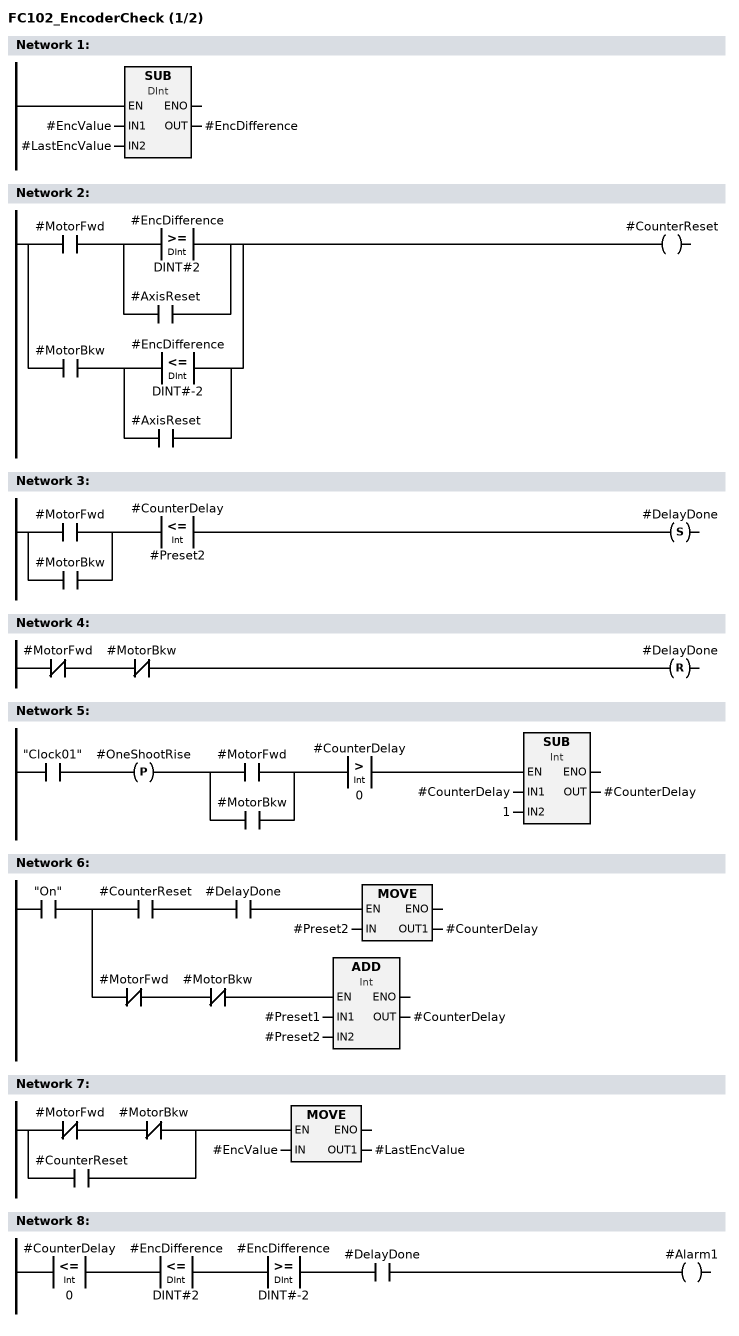
   RUNG wire#powerrail
      { S7_Templates := "SrcType := DInt"; S7_GenerateENO := "TRUE" } Sub(in1 := #EncValue, in2 := #LastEncValue, out => #EncDifference)
   END_RUNG
   // the same network as SCL:
   #EncDifference := #EncValue - #LastEncValue;
END_REGION

REGION Network 2
   RUNG wire#powerrail
      Contact( #MotorFwd )
      wire#w1
      { S7_Templates := "SrcType := DInt" } GE_Contact(in1 := #EncDifference, in2 := DINT#2)
      wire#w2
      Coil( #CounterReset )
   END_RUNG
   RUNG wire#w1
      Contact( #AxisReset )
   END_RUNG wire#w2
   RUNG wire#powerrail
      Contact( #MotorBkw )
      wire#w3
      { S7_Templates := "SrcType := DInt" } LE_Contact(in1 := #EncDifference, in2 := DINT#-2)
   END_RUNG wire#w2
   RUNG wire#w3
      Contact( #AxisReset )
   END_RUNG wire#w2
   // the same network as SCL:
   #CounterReset := (#MotorFwd AND ((#EncDifference >= DINT#2) OR #AxisReset)) OR (#MotorBkw AND ((#EncDifference <= DINT#-2) OR #AxisReset));
END_REGION

REGION Network 3
   RUNG wire#powerrail
      Contact( #MotorFwd )
      wire#w1
      { S7_Templates := "SrcType := Int" } LE_Contact(in1 := #CounterDelay, in2 := #Preset2)
      S_Coil( #DelayDone )
   END_RUNG
   RUNG wire#powerrail
      Contact( #MotorBkw )
   END_RUNG wire#w1
   // the same network as SCL:
   IF (#MotorFwd OR #MotorBkw) AND (#CounterDelay <= #Preset2) THEN #DelayDone := TRUE; END_IF;
END_REGION

REGION Network 4
   RUNG wire#powerrail
      I_Contact( #MotorFwd )
      I_Contact( #MotorBkw )
      R_Coil( #DelayDone )
   END_RUNG
   // the same network as SCL:
   IF NOT #MotorFwd AND NOT #MotorBkw THEN #DelayDone := FALSE; END_IF;
END_REGION

REGION Network 5
   RUNG wire#powerrail
      Contact( "Clock01" )
      P_Trig( #OneShootRise )
      wire#w1
      Contact( #MotorFwd )
      wire#w2
      { S7_Templates := "SrcType := Int" } GT_Contact(in1 := #CounterDelay, in2 := 0)
      { S7_Templates := "SrcType := Int"; S7_GenerateENO := "TRUE" } Sub(in1 := #CounterDelay, in2 := 1, out => #CounterDelay)
   END_RUNG
   RUNG wire#w1
      Contact( #MotorBkw )
   END_RUNG wire#w2
   // the same network as SCL:
   #_w1 := "Clock01" AND NOT #OneShootRise;   // rising edge
   #OneShootRise := "Clock01";
   IF #_w1 AND (#MotorFwd OR #MotorBkw) AND (#CounterDelay > 0) THEN
       #CounterDelay := #CounterDelay - 1;
   END_IF;
END_REGION

REGION Network 6
   RUNG wire#powerrail
      Contact( "On" )
      wire#w1
      Contact( #CounterReset )
      Contact( #DelayDone )
      { S7_GenerateENO := "TRUE" } Move(in := #Preset2, out1 => #CounterDelay)
   END_RUNG
   RUNG wire#w1
      I_Contact( #MotorFwd )
      I_Contact( #MotorBkw )
      { S7_Templates := "SrcType := Int"; S7_GenerateENO := "TRUE" } Add(in1 := #Preset1, in2 := #Preset2, out => #CounterDelay)
   END_RUNG
   // the same network as SCL:
   IF "On" AND #CounterReset AND #DelayDone THEN #CounterDelay := #Preset2; END_IF;
   IF "On" AND NOT #MotorFwd AND NOT #MotorBkw THEN #CounterDelay := #Preset1 + #Preset2; END_IF;
END_REGION

REGION Network 7
   RUNG wire#powerrail
      I_Contact( #MotorFwd )
      I_Contact( #MotorBkw )
      wire#w1
      { S7_GenerateENO := "TRUE" } Move(in := #EncValue, out1 => #LastEncValue)
   END_RUNG
   RUNG wire#powerrail
      Contact( #CounterReset )
   END_RUNG wire#w1
   // the same network as SCL:
   IF (NOT #MotorFwd AND NOT #MotorBkw) OR #CounterReset THEN #LastEncValue := #EncValue; END_IF;
END_REGION

REGION Network 8
   RUNG wire#powerrail
      { S7_Templates := "SrcType := Int" } LE_Contact(in1 := #CounterDelay, in2 := 0)
      { S7_Templates := "SrcType := DInt" } LE_Contact(in1 := #EncDifference, in2 := DINT#2)
      { S7_Templates := "SrcType := DInt" } GE_Contact(in1 := #EncDifference, in2 := DINT#-2)
      Contact( #DelayDone )
      Coil( #Alarm1 )
   END_RUNG
   // the same network as SCL:
   #Alarm1 := (#CounterDelay <= 0) AND (#EncDifference <= DINT#2) AND (#EncDifference >= DINT#-2) AND #DelayDone;
END_REGION

REGION Network 9
